LIN {X 0,Y 412.536,Z 861.906,A -85,B 0,C 180,E1 10223.476,E2 10223.476} C_VEL
LIN {X 0,Y 403.903,Z 849.532,A -85,B 0,C 180,E1 10225.593,E2 10225.593} C_VEL
LIN {X 0,Y 401.209,Z 844.898,A -85,B 0,C 180,E1 10226.312,E2 10226.312} C_VEL
LIN {X 0,Y 401.09,Z 843.44,A -85,B 0,C 180,E1 10226.508,E2 10226.508} C_VEL
LIN {X 0,Y 401.209,Z 843.44,A -85,B 0,C 180,E1 10233.172,E2 10233.172} C_VEL
LIN {X 0,Y 401.536,Z 843.44,A -85,B 0,C 180,E1 10240.232,E2 10240.232} C_VEL
LIN {X 0,Y 401.88,Z 843.44,A -85,B 0,C 180,E1 10246.981,E2 10246.981} C_VEL
LIN {X 0,Y 402.092,Z 843.44,A -85,B 0,C 180,E1 10253.536,E2 10253.536} C_VEL
LIN {X 0,Y 402.38,Z 843.44,A -85,B 0,C 180,E1 10260,E2 10260} C_VEL
LIN {X 0,Y 402.145,Z 843.44,A -85,B 0,C 180,E1 10266.464,E2 10266.464} C_VEL
LIN {X 0,Y 401.805,Z 843.44,A -85,B 0,C 180,E1 10273.022,E2 10273.022} C_VEL
LIN {X 0,Y 401.458,Z 843.44,A -85,B 0,C 180,E1 10279.998,E2 10279.998} C_VEL
LIN {X 0,Y 401.24,Z 843.44,A -85,B 0,C 180,E1 10286.827,E2 10286.827} C_VEL
LIN {X 0,Y 401.092,Z 844.186,A -85,B 0,C 180,E1 10293.067,E2 10293.067} C_VEL
LIN {X 0,Y 403.743,Z 849.357,A -85,B 0,C 180,E1 10293.796,E2 10293.796} C_VEL
LIN {X 0,Y 414.864,Z 865.253,A -85,B 0,C 180,E1 10296.457,E2 10296.457} C_VEL
LIN {X 0,Y 433.595,Z 895.537,A -85,B 0,C 180,E1 10300.541,E2 10300.541} C_VEL
LIN {X 0,Y 446.77,Z 923.801,A -85,B 0,C 180,E1 10303.625,E2 10303.625} C_VEL
LIN {X 0,Y 441.038,Z 966.249,A -85,B 0,C 180,E1 10305.53,E2 10305.53} C_VEL
LIN {X 0,Y 433.9,Z 1006.868,A -85,B 0,C 180,E1 10308.269,E2 10308.269} C_VEL
LIN {X 0,Y 425.996,Z 1044.808,A -85,B 0,C 180,E1 10311.841,E2 10311.841} C_VEL
LIN {X 0,Y 418.385,Z 1078.926,A -85,B 0,C 180,E1 10316.189,E2 10316.189} C_VEL
LIN {X 0,Y 411.832,Z 1108.737,A -85,B 0,C 180,E1 10321.255,E2 10321.255} C_VEL
LIN {X 0,Y 406.944,Z 1134.205,A -85,B 0,C 180,E1 10327.086,E2 10327.086} C_VEL
LIN {X 0,Y 404.04,Z 1153.414,A -85,B 0,C 180,E1 10333.175,E2 10333.175} C_VEL
LIN {X 0,Y 403.787,Z 1155.866,A -85,B 0,C 180,E1 10334.164,E2 10334.164} C_VEL
LIN {X 0,Y 400.89,Z 1159.99,A -85,B 0,C 180,E1 10335.894,E2 10335.894} C_VEL
LIN {X 0,Y 395.067,Z 1165.147,A -85,B 0,C 180,E1 10338.532,E2 10338.532} C_VEL
LIN {X 0,Y 394.935,Z 1165.692,A -85,B 0,C 180,E1 10338.841,E2 10338.841} C_VEL
LIN {X 0,Y 394.47,Z 1172.146,A -85,B 0,C 180,E1 10344.029,E2 10344.029} C_VEL
LIN {X 0,Y 394.523,Z 1174.816,A -85,B 0,C 180,E1 10350,E2 10350} C_VEL
LIN {X 0,Y 394.535,Z 1173.409,A -85,B 0,C 180,E1 10354.387,E2 10354.387} C_VEL
LIN {X 0,Y 394.794,Z 1167.57,A -85,B 0,C 180,E1 10359.905,E2 10359.905} C_VEL
LIN {X 0,Y 395.707,Z 1157.209,A -85,B 0,C 180,E1 10365.483,E2 10365.483} C_VEL
LIN {X 0,Y 398.3,Z 1139.989,A -85,B 0,C 180,E1 10371.636,E2 10371.636} C_VEL
LIN {X 0,Y 402.939,Z 1115.912,A -85,B 0,C 180,E1 10377.744,E2 10377.744} C_VEL
LIN {X 0,Y 409.269,Z 1088.112,A -85,B 0,C 180,E1 10382.969,E2 10382.969} C_VEL
LIN {X 0,Y 417.087,Z 1054.957,A -85,B 0,C 180,E1 10387.641,E2 10387.641} C_VEL
LIN {X 0,Y 425.41,Z 1017.824,A -85,B 0,C 180,E1 10391.513,E2 10391.513} C_VEL
LIN {X 0,Y 433.374,Z 977.18,A -85,B 0,C 180,E1 10394.553,E2 10394.553} C_VEL
LIN {X 0,Y 439.964,Z 934.17,A -85,B 0,C 180,E1 10396.732,E2 10396.732} C_VEL
LIN {X 0,Y 440.381,Z 925.23,A -85,B 0,C 180,E1 10397.161,E2 10397.161} C_VEL
LIN {X 0,Y 425.642,Z 894.694,A -85,B 0,C 180,E1 10400.751,E2 10400.751} C_VEL
LIN {X 0,Y 409.009,Z 867.964,A -85,B 0,C 180,E1 10404.593,E2 10404.593} C_VEL
LIN {X 0,Y 396.315,Z 849.753,A -85,B 0,C 180,E1 10407.836,E2 10407.836} C_VEL
LIN {X 0,Y 393.263,Z 844.634,A -85,B 0,C 180,E1 10408.718,E2 10408.718} C_VEL
LIN {X 0,Y 393.154,Z 843.44,A -85,B 0,C 180,E1 10408.818,E2 10408.818} C_VEL
LIN {X 0,Y 393.359,Z 843.44,A -85,B 0,C 180,E1 10415.041,E2 10415.041} C_VEL
LIN {X 0,Y 393.632,Z 843.44,A -85,B 0,C 180,E1 10422.141,E2 10422.141} C_VEL
LIN {X 0,Y 393.836,Z 843.44,A -85,B 0,C 180,E1 10428.955,E2 10428.955} C_VEL
LIN {X 0,Y 394.243,Z 843.44,A -85,B 0,C 180,E1 10435.61,E2 10435.61} C_VEL
LIN {X 0,Y 394.337,Z 843.44,A -85,B 0,C 180,E1 10442.193,E2 10442.193} C_VEL
LIN {X 0,Y 394.018,Z 843.44,A -85,B 0,C 180,E1 10448.811,E2 10448.811} C_VEL
LIN {X 0,Y 393.774,Z 843.44,A -85,B 0,C 180,E1 10455.559,E2 10455.559} C_VEL
LIN {X 0,Y 393.41,Z 843.44,A -85,B 0,C 180,E1 10462.989,E2 10462.989} C_VEL
LIN {X 0,Y 393.294,Z 843.44,A -85,B 0,C 180,E1 10469.919,E2 10469.919} C_VEL
LIN {X 0,Y 393.33,Z 843.44,A -85,B 0,C 180,E1 10471.727,E2 10471.727} C_VEL
LIN {X 0,Y 395.292,Z 848.705,A -85,B 0,C 180,E1 10472.377,E2 10472.377} C_VEL
LIN {X 0,Y 398.335,Z 852.335,A -85,B 0,C 180,E1 10473.186,E2 10473.186} C_VEL
LIN {X 0,Y 414.19,Z 876.466,A -85,B 0,C 180,E1 10477.277,E2 10477.277} C_VEL
LIN {X 0,Y 429.429,Z 905.007,A -85,B 0,C 180,E1 10481.288,E2 10481.288} C_VEL
LIN {X 0,Y 438.439,Z 927.966,A -85,B 0,C 180,E1 10484.052,E2 10484.052} C_VEL
LIN {X 0,Y 431.611,Z 968.432,A -85,B 0,C 180,E1 10486.494,E2 10486.494} C_VEL
LIN {X 0,Y 423.482,Z 1006.655,A -85,B 0,C 180,E1 10489.77,E2 10489.77} C_VEL
LIN {X 0,Y 415.09,Z 1041.89,A -85,B 0,C 180,E1 10493.94,E2 10493.94} C_VEL
LIN {X 0,Y 407.221,Z 1073.607,A -85,B 0,C 180,E1 10499.059,E2 10499.059} C_VEL
LIN {X 0,Y 401.372,Z 1098.435,A -85,B 0,C 180,E1 10504.459,E2 10504.459} C_VEL
LIN {X 0,Y 397.287,Z 1119.022,A -85,B 0,C 180,E1 10510.615,E2 10510.615} C_VEL
LIN {X 0,Y 395.387,Z 1133.199,A -85,B 0,C 180,E1 10516.762,E2 10516.762} C_VEL
LIN {X 0,Y 394.56,Z 1141.136,A -85,B 0,C 180,E1 10522.307,E2 10522.307} C_VEL
LIN {X 0,Y 394.48,Z 1144.909,A -85,B 0,C 180,E1 10527.807,E2 10527.807} C_VEL
LIN {X 0,Y 394.579,Z 1144.88,A -85,B 0,C 180,E1 10532.192,E2 10532.192} C_VEL
LIN {X 0,Y 394.625,Z 1141.038,A -85,B 0,C 180,E1 10537.691,E2 10537.691} C_VEL
LIN {X 0,Y 395.504,Z 1132.152,A -85,B 0,C 180,E1 10543.672,E2 10543.672} C_VEL
LIN {X 0,Y 397.375,Z 1118.609,A -85,B 0,C 180,E1 10549.449,E2 10549.449} C_VEL
LIN {X 0,Y 401.431,Z 1098.022,A -85,B 0,C 180,E1 10555.559,E2 10555.559} C_VEL
LIN {X 0,Y 407.649,Z 1071.682,A -85,B 0,C 180,E1 10561.214,E2 10561.214} C_VEL
LIN {X 0,Y 415.306,Z 1041.141,A -85,B 0,C 180,E1 10566.063,E2 10566.063} C_VEL
LIN {X 0,Y 423.441,Z 1006.999,A -85,B 0,C 180,E1 10570.1,E2 10570.1} C_VEL
LIN {X 0,Y 431.425,Z 969.351,A -85,B 0,C 180,E1 10573.35,E2 10573.35} C_VEL
LIN {X 0,Y 438.451,Z 927.099,A -85,B 0,C 180,E1 10575.909,E2 10575.909} C_VEL
LIN {X 0,Y 424.695,Z 895.119,A -85,B 0,C 180,E1 10579.911,E2 10579.911} C_VEL
LIN {X 0,Y 408.354,Z 867.268,A -85,B 0,C 180,E1 10584.097,E2 10584.097} C_VEL
LIN {X 0,Y 396.169,Z 849.642,A -85,B 0,C 180,E1 10587.277,E2 10587.277} C_VEL
LIN {X 0,Y 393.281,Z 844.581,A -85,B 0,C 180,E1 10588.118,E2 10588.118} C_VEL
LIN {X 0,Y 393.187,Z 843.44,A -85,B 0,C 180,E1 10588.384,E2 10588.384} C_VEL
LIN {X 0,Y 393.352,Z 843.44,A -85,B 0,C 180,E1 10595.041,E2 10595.041} C_VEL
LIN {X 0,Y 393.712,Z 843.44,A -85,B 0,C 180,E1 10602.145,E2 10602.145} C_VEL
LIN {X 0,Y 393.997,Z 843.44,A -85,B 0,C 180,E1 10608.96,E2 10608.96} C_VEL
LIN {X 0,Y 394.278,Z 843.44,A -85,B 0,C 180,E1 10615.61,E2 10615.61} C_VEL
LIN {X 0,Y 394.482,Z 843.44,A -85,B 0,C 180,E1 10622.192,E2 10622.192} C_VEL
LIN {X 0,Y 394.04,Z 843.44,A -85,B 0,C 180,E1 10628.811,E2 10628.811} C_VEL
LIN {X 0,Y 393.727,Z 843.44,A -85,B 0,C 180,E1 10635.562,E2 10635.562} C_VEL
LIN {X 0,Y 393.413,Z 843.44,A -85,B 0,C 180,E1 10642.991,E2 10642.991} C_VEL
LIN {X 0,Y 393.194,Z 843.44,A -85,B 0,C 180,E1 10649.927,E2 10649.927} C_VEL
LIN {X 0,Y 393.158,Z 843.44,A -85,B 0,C 180,E1 10651.238,E2 10651.238} C_VEL
LIN {X 0,Y 395.313,Z 848.816,A -85,B 0,C 180,E1 10651.927,E2 10651.927} C_VEL
LIN {X 0,Y 398.159,Z 852.24,A -85,B 0,C 180,E1 10652.683,E2 10652.683} C_VEL
LIN {X 0,Y 417.725,Z 881.071,A -85,B 0,C 180,E1 10657.445,E2 10657.445} C_VEL
LIN {X 0,Y 434.757,Z 912.535,A -85,B 0,C 180,E1 10661.424,E2 10661.424} C_VEL
LIN {X 0,Y 440.859,Z 927.31,A -85,B 0,C 180,E1 10663.022,E2 10663.022} C_VEL
LIN {X 0,Y 435.214,Z 966.606,A -85,B 0,C 180,E1 10664.827,E2 10664.827} C_VEL
LIN {X 0,Y 427.789,Z 1006.919,A -85,B 0,C 180,E1 10667.575,E2 10667.575} C_VEL
LIN {X 0,Y 419.756,Z 1043.593,A -85,B 0,C 180,E1 10671.047,E2 10671.047} C_VEL
LIN {X 0,Y 411.516,Z 1078.613,A -85,B 0,C 180,E1 10675.546,E2 10675.546} C_VEL
LIN {X 0,Y 404.609,Z 1108.428,A -85,B 0,C 180,E1 10680.692,E2 10680.692} C_VEL
LIN {X 0,Y 399.343,Z 1133.895,A -85,B 0,C 180,E1 10686.624,E2 10686.624} C_VEL
LIN {X 0,Y 396.253,Z 1153.109,A -85,B 0,C 180,E1 10692.835,E2 10692.835} C_VEL
LIN {X 0,Y 394.935,Z 1165.692,A -85,B 0,C 180,E1 10698.841,E2 10698.841} C_VEL
LIN {X 0,Y 392.233,Z 1168.533,A -85,B 0,C 180,E1 10700.665,E2 10700.665} C_VEL
LIN {X 0,Y 386.689,Z 1171.487,A -85,B 0,C 180,E1 10703.446,E2 10703.446} C_VEL
LIN {X 0,Y 386.568,Z 1171.734,A -85,B 0,C 180,E1 10703.771,E2 10703.771} C_VEL
LIN {X 0,Y 386.572,Z 1174.166,A -85,B 0,C 180,E1 10707.763,E2 10707.763} C_VEL
LIN {X 0,Y 386.751,Z 1174.172,A -85,B 0,C 180,E1 10712.236,E2 10712.236} C_VEL
LIN {X 0,Y 386.706,Z 1170.117,A -85,B 0,C 180,E1 10717.85,E2 10717.85} C_VEL
LIN {X 0,Y 387.441,Z 1161.671,A -85,B 0,C 180,E1 10723.515,E2 10723.515} C_VEL
LIN {X 0,Y 389.437,Z 1146.627,A -85,B 0,C 180,E1 10729.819,E2 10729.819} C_VEL
LIN {X 0,Y 393.295,Z 1126.005,A -85,B 0,C 180,E1 10735.858,E2 10735.858} C_VEL
LIN {X 0,Y 399.461,Z 1099.256,A -85,B 0,C 180,E1 10741.611,E2 10741.611} C_VEL
LIN {X 0,Y 407.687,Z 1066.369,A -85,B 0,C 180,E1 10746.83,E2 10746.83} C_VEL
LIN {X 0,Y 416.394,Z 1030.711,A -85,B 0,C 180,E1 10750.997,E2 10750.997} C_VEL
LIN {X 0,Y 424.702,Z 992.738,A -85,B 0,C 180,E1 10754.24,E2 10754.24} C_VEL
LIN {X 0,Y 431.692,Z 953.938,A -85,B 0,C 180,E1 10756.581,E2 10756.581} C_VEL
LIN {X 0,Y 434.563,Z 928.474,A -85,B 0,C 180,E1 10757.795,E2 10757.795} C_VEL
LIN {X 0,Y 420.517,Z 898.817,A -85,B 0,C 180,E1 10761.43,E2 10761.43} C_VEL
LIN {X 0,Y 404.771,Z 873.027,A -85,B 0,C 180,E1 10765.284,E2 10765.284} C_VEL
LIN {X 0,Y 392.687,Z 855.818,A -85,B 0,C 180,E1 10768.473,E2 10768.473} C_VEL
LIN {X 0,Y 388.57,Z 849.833,A -85,B 0,C 180,E1 10769.679,E2 10769.679} C_VEL
LIN {X 0,Y 385.501,Z 845.356,A -85,B 0,C 180,E1 10770.626,E2 10770.626} C_VEL
LIN {X 0,Y 385.254,Z 843.44,A -85,B 0,C 180,E1 10770.85,E2 10770.85} C_VEL
LIN {X 0,Y 385.514,Z 843.44,A -85,B 0,C 180,E1 10776.957,E2 10776.957} C_VEL
LIN {X 0,Y 385.745,Z 843.44,A -85,B 0,C 180,E1 10784.108,E2 10784.108} C_VEL
LIN {X 0,Y 386.034,Z 843.44,A -85,B 0,C 180,E1 10791.004,E2 10791.004} C_VEL
LIN {X 0,Y 386.575,Z 843.44,A -85,B 0,C 180,E1 10797.763,E2 10797.763} C_VEL
LIN {X 0,Y 386.362,Z 843.44,A -85,B 0,C 180,E1 10804.48,E2 10804.48} C_VEL
LIN {X 0,Y 386.024,Z 843.44,A -85,B 0,C 180,E1 10811.271,E2 10811.271} C_VEL
LIN {X 0,Y 385.695,Z 843.44,A -85,B 0,C 180,E1 10818.239,E2 10818.239} C_VEL
LIN {X 0,Y 385.366,Z 843.44,A -85,B 0,C 180,E1 10825.758,E2 10825.758} C_VEL
LIN {X 0,Y 385.373,Z 843.44,A -85,B 0,C 180,E1 10829.752,E2 10829.752} C_VEL
LIN {X 0,Y 387.473,Z 848.827,A -85,B 0,C 180,E1 10830.491,E2 10830.491} C_VEL
LIN {X 0,Y 390.513,Z 852.225,A -85,B 0,C 180,E1 10831.366,E2 10831.366} C_VEL
LIN {X 0,Y 406.881,Z 876.641,A -85,B 0,C 180,E1 10835.891,E2 10835.891} C_VEL
LIN {X 0,Y 422.767,Z 906.139,A -85,B 0,C 180,E1 10840.296,E2 10840.296} C_VEL
LIN {X 0,Y 432.571,Z 930.558,A -85,B 0,C 180,E1 10843.415,E2 10843.415} C_VEL
LIN {X 0,Y 425.827,Z 968.818,A -85,B 0,C 180,E1 10845.759,E2 10845.759} C_VEL
LIN {X 0,Y 417.032,Z 1008.301,A -85,B 0,C 180,E1 10849.19,E2 10849.19} C_VEL
LIN {X 0,Y 408.103,Z 1043.878,A -85,B 0,C 180,E1 10853.513,E2 10853.513} C_VEL
LIN {X 0,Y 400.196,Z 1073.911,A -85,B 0,C 180,E1 10858.454,E2 10858.454} C_VEL
LIN {X 0,Y 394.079,Z 1098.735,A -85,B 0,C 180,E1 10863.951,E2 10863.951} C_VEL
LIN {X 0,Y 389.646,Z 1119.254,A -85,B 0,C 180,E1 10870.192,E2 10870.192} C_VEL
LIN {X 0,Y 387.567,Z 1133.498,A -85,B 0,C 180,E1 10876.49,E2 10876.49} C_VEL
LIN {X 0,Y 386.683,Z 1141.433,A -85,B 0,C 180,E1 10882.149,E2 10882.149} C_VEL
LIN {X 0,Y 386.581,Z 1145.206,A -85,B 0,C 180,E1 10887.763,E2 10887.763} C_VEL
LIN {X 0,Y 386.678,Z 1145.177,A -85,B 0,C 180,E1 10892.236,E2 10892.236} C_VEL
LIN {X 0,Y 386.745,Z 1141.337,A -85,B 0,C 180,E1 10897.849,E2 10897.849} C_VEL
LIN {X 0,Y 387.634,Z 1133.323,A -85,B 0,C 180,E1 10903.507,E2 10903.507} C_VEL
LIN {X 0,Y 389.689,Z 1119.028,A -85,B 0,C 180,E1 10909.805,E2 10909.805} C_VEL
LIN {X 0,Y 394.081,Z 1098.332,A -85,B 0,C 180,E1 10916.071,E2 10916.071} C_VEL
LIN {X 0,Y 400.688,Z 1071.993,A -85,B 0,C 180,E1 10921.819,E2 10921.819} C_VEL
LIN {X 0,Y 408.657,Z 1041.936,A -85,B 0,C 180,E1 10926.668,E2 10926.668} C_VEL
LIN {X 0,Y 417.257,Z 1007.566,A -85,B 0,C 180,E1 10930.786,E2 10930.786} C_VEL
LIN {X 0,Y 425.671,Z 969.676,A -85,B 0,C 180,E1 10934.084,E2 10934.084} C_VEL
LIN {X 0,Y 432.479,Z 930.241,A -85,B 0,C 180,E1 10936.527,E2 10936.527} C_VEL
LIN {X 0,Y 419.451,Z 899.303,A -85,B 0,C 180,E1 10940.567,E2 10940.567} C_VEL
LIN {X 0,Y 402.739,Z 869.859,A -85,B 0,C 180,E1 10945.135,E2 10945.135} C_VEL
LIN {X 0,Y 388.559,Z 849.846,A -85,B 0,C 180,E1 10949.081,E2 10949.081} C_VEL
LIN {X 0,Y 385.437,Z 844.892,A -85,B 0,C 180,E1 10950.056,E2 10950.056} C_VEL
LIN {X 0,Y 385.275,Z 843.44,A -85,B 0,C 180,E1 10950.366,E2 10950.366} C_VEL
LIN {X 0,Y 385.51,Z 843.44,A -85,B 0,C 180,E1 10956.958,E2 10956.958} C_VEL
LIN {X 0,Y 385.91,Z 843.44,A -85,B 0,C 180,E1 10964.115,E2 10964.115} C_VEL
LIN {X 0,Y 386.126,Z 843.44,A -85,B 0,C 180,E1 10971.007,E2 10971.007} C_VEL
LIN {X 0,Y 386.439,Z 843.44,A -85,B 0,C 180,E1 10977.762,E2 10977.762} C_VEL
LIN {X 0,Y 386.335,Z 843.44,A -85,B 0,C 180,E1 10984.481,E2 10984.481} C_VEL
LIN {X 0,Y 385.981,Z 843.44,A -85,B 0,C 180,E1 10991.272,E2 10991.272} C_VEL
LIN {X 0,Y 385.668,Z 843.44,A -85,B 0,C 180,E1 10998.241,E2 10998.241} C_VEL
LIN {X 0,Y 385.383,Z 843.44,A -85,B 0,C 180,E1 11005.512,E2 11005.512} C_VEL
LIN {X 0,Y 385.302,Z 844.197,A -85,B 0,C 180,E1 11009.31,E2 11009.31} C_VEL
LIN {X 0,Y 388.071,Z 849.476,A -85,B 0,C 180,E1 11010.212,E2 11010.212} C_VEL
LIN {X 0,Y 390.458,Z 852.409,A -85,B 0,C 180,E1 11010.903,E2 11010.903} C_VEL
LIN {X 0,Y 407.64,Z 877.287,A -85,B 0,C 180,E1 11015.444,E2 11015.444} C_VEL
LIN {X 0,Y 424.478,Z 906.09,A -85,B 0,C 180,E1 11019.534,E2 11019.534} C_VEL
LIN {X 0,Y 434.994,Z 930.293,A -85,B 0,C 180,E1 11022.373,E2 11022.373} C_VEL
LIN {X 0,Y 428.859,Z 970.174,A -85,B 0,C 180,E1 11024.293,E2 11024.293} C_VEL
LIN {X 0,Y 421.471,Z 1008.185,A -85,B 0,C 180,E1 11026.964,E2 11026.964} C_VEL
LIN {X 0,Y 412.982,Z 1044.955,A -85,B 0,C 180,E1 11030.521,E2 11030.521} C_VEL
LIN {X 0,Y 404.635,Z 1078.785,A -85,B 0,C 180,E1 11034.963,E2 11034.963} C_VEL
LIN {X 0,Y 397.422,Z 1108.117,A -85,B 0,C 180,E1 11040.109,E2 11040.109} C_VEL
LIN {X 0,Y 391.775,Z 1133.585,A -85,B 0,C 180,E1 11046.145,E2 11046.145} C_VEL
LIN {X 0,Y 388.705,Z 1151.329,A -85,B 0,C 180,E1 11051.906,E2 11051.906} C_VEL
LIN {X 0,Y 387.252,Z 1163.986,A -85,B 0,C 180,E1 11057.801,E2 11057.801} C_VEL
LIN {X 0,Y 386.629,Z 1171.345,A -85,B 0,C 180,E1 11063.276,E2 11063.276} C_VEL
LIN {X 0,Y 386.568,Z 1171.734,A -85,B 0,C 180,E1 11063.771,E2 11063.771} C_VEL
LIN {X 0,Y 383.964,Z 1173.1,A -85,B 0,C 180,E1 11065.669,E2 11065.669} C_VEL
LIN {X 0,Y 378.708,Z 1174.007,A -85,B 0,C 180,E1 11068.538,E2 11068.538} C_VEL
LIN {X 0,Y 378.626,Z 1174.048,A -85,B 0,C 180,E1 11068.871,E2 11068.871} C_VEL
LIN {X 0,Y 378.845,Z 1173.876,A -85,B 0,C 180,E1 11072.283,E2 11072.283} C_VEL
LIN {X 0,Y 378.821,Z 1169.818,A -85,B 0,C 180,E1 11078.015,E2 11078.015} C_VEL
LIN {X 0,Y 379.571,Z 1161.367,A -85,B 0,C 180,E1 11083.8,E2 11083.8} C_VEL
LIN {X 0,Y 381.744,Z 1146.32,A -85,B 0,C 180,E1 11090.236,E2 11090.236} C_VEL
LIN {X 0,Y 386.289,Z 1124.406,A -85,B 0,C 180,E1 11096.719,E2 11096.719} C_VEL
LIN {X 0,Y 392.864,Z 1097.403,A -85,B 0,C 180,E1 11102.531,E2 11102.531} C_VEL
LIN {X 0,Y 401.145,Z 1066.056,A -85,B 0,C 180,E1 11107.534,E2 11107.534} C_VEL
LIN {X 0,Y 410.439,Z 1029.58,A -85,B 0,C 180,E1 11111.828,E2 11111.828} C_VEL
LIN {X 0,Y 419.296,Z 990.383,A -85,B 0,C 180,E1 11115.164,E2 11115.164} C_VEL
LIN {X 0,Y 426.852,Z 949.888,A -85,B 0,C 180,E1 11117.556,E2 11117.556} C_VEL
LIN {X 0,Y 428.835,Z 931.703,A -85,B 0,C 180,E1 11118.443,E2 11118.443} C_VEL
LIN {X 0,Y 414.799,Z 901.66,A -85,B 0,C 180,E1 11122.294,E2 11122.294} C_VEL
LIN {X 0,Y 398.816,Z 875.264,A -85,B 0,C 180,E1 11126.451,E2 11126.451} C_VEL
LIN {X 0,Y 385.116,Z 856.082,A -85,B 0,C 180,E1 11130.331,E2 11130.331} C_VEL
LIN {X 0,Y 381.085,Z 850.146,A -85,B 0,C 180,E1 11131.63,E2 11131.63} C_VEL
LIN {X 0,Y 377.608,Z 845.437,A -85,B 0,C 180,E1 11132.803,E2 11132.803} C_VEL
LIN {X 0,Y 377.364,Z 843.44,A -85,B 0,C 180,E1 11133.105,E2 11133.105} C_VEL
LIN {X 0,Y 377.637,Z 843.44,A -85,B 0,C 180,E1 11138.923,E2 11138.923} C_VEL
LIN {X 0,Y 377.882,Z 843.44,A -85,B 0,C 180,E1 11146.137,E2 11146.137} C_VEL
LIN {X 0,Y 378.33,Z 843.44,A -85,B 0,C 180,E1 11153.128,E2 11153.128} C_VEL
LIN {X 0,Y 378.628,Z 843.44,A -85,B 0,C 180,E1 11160,E2 11160} C_VEL
LIN {X 0,Y 378.323,Z 843.44,A -85,B 0,C 180,E1 11166.872,E2 11166.872} C_VEL
LIN {X 0,Y 378.021,Z 843.44,A -85,B 0,C 180,E1 11173.857,E2 11173.857} C_VEL
LIN {X 0,Y 377.633,Z 843.44,A -85,B 0,C 180,E1 11181.077,E2 11181.077} C_VEL
LIN {X 0,Y 377.427,Z 843.515,A -85,B 0,C 180,E1 11187.549,E2 11187.549} C_VEL
LIN {X 0,Y 379.422,Z 848.673,A -85,B 0,C 180,E1 11188.331,E2 11188.331} C_VEL
LIN {X 0,Y 382.7,Z 852.12,A -85,B 0,C 180,E1 11189.367,E2 11189.367} C_VEL
LIN {X 0,Y 397.567,Z 873.908,A -85,B 0,C 180,E1 11193.826,E2 11193.826} C_VEL
LIN {X 0,Y 412.618,Z 900.242,A -85,B 0,C 180,E1 11198.189,E2 11198.189} C_VEL
LIN {X 0,Y 424.836,Z 928.377,A -85,B 0,C 180,E1 11202.099,E2 11202.099} C_VEL
LIN {X 0,Y 426.507,Z 934.531,A -85,B 0,C 180,E1 11202.833,E2 11202.833} C_VEL
LIN {X 0,Y 419.384,Z 972.555,A -85,B 0,C 180,E1 11205.26,E2 11205.26} C_VEL
LIN {X 0,Y 410.623,Z 1009.825,A -85,B 0,C 180,E1 11208.586,E2 11208.586} C_VEL
LIN {X 0,Y 401.559,Z 1044.313,A -85,B 0,C 180,E1 11212.843,E2 11212.843} C_VEL
LIN {X 0,Y 393.263,Z 1074.214,A -85,B 0,C 180,E1 11217.831,E2 11217.831} C_VEL
LIN {X 0,Y 386.735,Z 1099.222,A -85,B 0,C 180,E1 11223.472,E2 11223.472} C_VEL
LIN {X 0,Y 382.038,Z 1119.556,A -85,B 0,C 180,E1 11229.78,E2 11229.78} C_VEL
LIN {X 0,Y 379.777,Z 1133.797,A -85,B 0,C 180,E1 11236.207,E2 11236.207} C_VEL
LIN {X 0,Y 378.804,Z 1141.731,A -85,B 0,C 180,E1 11241.985,E2 11241.985} C_VEL
LIN {X 0,Y 378.682,Z 1145.502,A -85,B 0,C 180,E1 11247.716,E2 11247.716} C_VEL
LIN {X 0,Y 378.777,Z 1145.474,A -85,B 0,C 180,E1 11252.283,E2 11252.283} C_VEL
LIN {X 0,Y 378.889,Z 1141.636,A -85,B 0,C 180,E1 11258.013,E2 11258.013} C_VEL
LIN {X 0,Y 379.827,Z 1133.626,A -85,B 0,C 180,E1 11263.79,E2 11263.79} C_VEL
LIN {X 0,Y 382.049,Z 1119.335,A -85,B 0,C 180,E1 11270.219,E2 11270.219} C_VEL
LIN {X 0,Y 386.505,Z 1099.673,A -85,B 0,C 180,E1 11276.324,E2 11276.324} C_VEL
LIN {X 0,Y 393.373,Z 1073.813,A -85,B 0,C 180,E1 11282.158,E2 11282.158} C_VEL
LIN {X 0,Y 402.097,Z 1042.502,A -85,B 0,C 180,E1 11287.324,E2 11287.324} C_VEL
LIN {X 0,Y 411.179,Z 1007.885,A -85,B 0,C 180,E1 11291.519,E2 11291.519} C_VEL
LIN {X 0,Y 419.968,Z 969.983,A -85,B 0,C 180,E1 11294.842,E2 11294.842} C_VEL
LIN {X 0,Y 426.377,Z 933.046,A -85,B 0,C 180,E1 11297.206,E2 11297.206} C_VEL
LIN {X 0,Y 413.914,Z 902.607,A -85,B 0,C 180,E1 11301.33,E2 11301.33} C_VEL
LIN {X 0,Y 398.105,Z 874.851,A -85,B 0,C 180,E1 11305.899,E2 11305.899} C_VEL
LIN {X 0,Y 385.288,Z 856.281,A -85,B 0,C 180,E1 11309.677,E2 11309.677} C_VEL
LIN {X 0,Y 380.858,Z 850.005,A -85,B 0,C 180,E1 11311.092,E2 11311.092} C_VEL
LIN {X 0,Y 377.529,Z 844.979,A -85,B 0,C 180,E1 11312.234,E2 11312.234} C_VEL
LIN {X 0,Y 377.349,Z 843.44,A -85,B 0,C 180,E1 11312.392,E2 11312.392} C_VEL
LIN {X 0,Y 377.644,Z 843.44,A -85,B 0,C 180,E1 11318.924,E2 11318.924} C_VEL
LIN {X 0,Y 378.07,Z 843.44,A -85,B 0,C 180,E1 11326.145,E2 11326.145} C_VEL
LIN {X 0,Y 378.328,Z 843.44,A -85,B 0,C 180,E1 11333.128,E2 11333.128} C_VEL
LIN {X 0,Y 378.673,Z 843.44,A -85,B 0,C 180,E1 11340,E2 11340} C_VEL
LIN {X 0,Y 378.402,Z 843.44,A -85,B 0,C 180,E1 11346.871,E2 11346.871} C_VEL
LIN {X 0,Y 377.956,Z 843.44,A -85,B 0,C 180,E1 11353.86,E2 11353.86} C_VEL
LIN {X 0,Y 377.622,Z 843.44,A -85,B 0,C 180,E1 11361.078,E2 11361.078} C_VEL
LIN {X 0,Y 377.42,Z 844.229,A -85,B 0,C 180,E1 11367.131,E2 11367.131} C_VEL
LIN {X 0,Y 380.045,Z 849.339,A -85,B 0,C 180,E1 11368.084,E2 11368.084} C_VEL
LIN {X 0,Y 382.648,Z 852.309,A -85,B 0,C 180,E1 11368.91,E2 11368.91} C_VEL
LIN {X 0,Y 397.159,Z 872.998,A -85,B 0,C 180,E1 11373.133,E2 11373.133} C_VEL
LIN {X 0,Y 413.401,Z 899.125,A -85,B 0,C 180,E1 11377.361,E2 11377.361} C_VEL
LIN {X 0,Y 427.986,Z 929.72,A -85,B 0,C 180,E1 11381.324,E2 11381.324} C_VEL
LIN {X 0,Y 429.039,Z 934.674,A -85,B 0,C 180,E1 11381.764,E2 11381.764} C_VEL
LIN {X 0,Y 421.653,Z 978.391,A -85,B 0,C 180,E1 11384.019,E2 11384.019} C_VEL
LIN {X 0,Y 412.864,Z 1019.432,A -85,B 0,C 180,E1 11387.198,E2 11387.198} C_VEL
LIN {X 0,Y 403.964,Z 1055.351,A -85,B 0,C 180,E1 11391.063,E2 11391.063} C_VEL
LIN {X 0,Y 395.033,Z 1089.295,A -85,B 0,C 180,E1 11396.036,E2 11396.036} C_VEL
LIN {X 0,Y 388.028,Z 1116.746,A -85,B 0,C 180,E1 11401.441,E2 11401.441} C_VEL
LIN {X 0,Y 382.955,Z 1140.091,A -85,B 0,C 180,E1 11407.688,E2 11407.688} C_VEL
LIN {X 0,Y 380.182,Z 1156.604,A -85,B 0,C 180,E1 11413.869,E2 11413.869} C_VEL
LIN {X 0,Y 379.018,Z 1166.97,A -85,B 0,C 180,E1 11419.679,E2 11419.679} C_VEL
LIN {X 0,Y 378.696,Z 1172.813,A -85,B 0,C 180,E1 11425.429,E2 11425.429} C_VEL
LIN {X 0,Y 378.626,Z 1174.048,A -85,B 0,C 180,E1 11428.871,E2 11428.871} C_VEL
LIN {X 0,Y 376.16,Z 1174.04,A -85,B 0,C 180,E1 11430.831,E2 11430.831} C_VEL
LIN {X 0,Y 370.82,Z 1172.766,A -85,B 0,C 180,E1 11434.122,E2 11434.122} C_VEL
LIN {X 0,Y 371.036,Z 1168.266,A -85,B 0,C 180,E1 11439.363,E2 11439.363} C_VEL
LIN {X 0,Y 372.167,Z 1157.538,A -85,B 0,C 180,E1 11445.884,E2 11445.884} C_VEL
LIN {X 0,Y 375.062,Z 1141.279,A -85,B 0,C 180,E1 11452.28,E2 11452.28} C_VEL
LIN {X 0,Y 380.011,Z 1119.297,A -85,B 0,C 180,E1 11458.458,E2 11458.458} C_VEL
LIN {X 0,Y 386.797,Z 1093.853,A -85,B 0,C 180,E1 11463.776,E2 11463.776} C_VEL
LIN {X 0,Y 395.109,Z 1063.973,A -85,B 0,C 180,E1 11468.502,E2 11468.502} C_VEL
LIN {X 0,Y 404.477,Z 1028.861,A -85,B 0,C 180,E1 11472.642,E2 11472.642} C_VEL
LIN {X 0,Y 413.669,Z 989.935,A -85,B 0,C 180,E1 11475.968,E2 11475.968} C_VEL
LIN {X 0,Y 421.657,Z 948.183,A -85,B 0,C 180,E1 11478.431,E2 11478.431} C_VEL
LIN {X 0,Y 423.436,Z 935.798,A -85,B 0,C 180,E1 11479.011,E2 11479.011} C_VEL
LIN {X 0,Y 410,Z 906.276,A -85,B 0,C 180,E1 11482.939,E2 11482.939} C_VEL
LIN {X 0,Y 395.064,Z 881.076,A -85,B 0,C 180,E1 11487.047,E2 11487.047} C_VEL
LIN {X 0,Y 381.653,Z 861.918,A -85,B 0,C 180,E1 11491.027,E2 11491.027} C_VEL
LIN {X 0,Y 377.311,Z 856.085,A -85,B 0,C 180,E1 11492.461,E2 11492.461} C_VEL
LIN {X 0,Y 373.359,Z 850.218,A -85,B 0,C 180,E1 11493.883,E2 11493.883} C_VEL
LIN {X 0,Y 369.785,Z 845.578,A -85,B 0,C 180,E1 11495.231,E2 11495.231} C_VEL
LIN {X 0,Y 369.521,Z 843.44,A -85,B 0,C 180,E1 11495.441,E2 11495.441} C_VEL
LIN {X 0,Y 369.774,Z 843.44,A -85,B 0,C 180,E1 11500.946,E2 11500.946} C_VEL
LIN {X 0,Y 370.042,Z 843.44,A -85,B 0,C 180,E1 11508.235,E2 11508.235} C_VEL
LIN {X 0,Y 370.506,Z 843.44,A -85,B 0,C 180,E1 11515.328,E2 11515.328} C_VEL
LIN {X 0,Y 370.751,Z 843.44,A -85,B 0,C 180,E1 11520,E2 11520} C_VEL
LIN {X 0,Y 370.392,Z 843.44,A -85,B 0,C 180,E1 11527.02,E2 11527.02} C_VEL
LIN {X 0,Y 370.095,Z 843.44,A -85,B 0,C 180,E1 11534.16,E2 11534.16} C_VEL
LIN {X 0,Y 369.693,Z 843.44,A -85,B 0,C 180,E1 11541.552,E2 11541.552} C_VEL
LIN {X 0,Y 369.519,Z 843.756,A -85,B 0,C 180,E1 11545.081,E2 11545.081} C_VEL
LIN {X 0,Y 371.586,Z 848.762,A -85,B 0,C 180,E1 11545.98,E2 11545.98} C_VEL
LIN {X 0,Y 374.98,Z 852.27,A -85,B 0,C 180,E1 11547.181,E2 11547.181} C_VEL
LIN {X 0,Y 389.017,Z 872.069,A -85,B 0,C 180,E1 11551.782,E2 11551.782} C_VEL
LIN {X 0,Y 404.476,Z 898.403,A -85,B 0,C 180,E1 11556.565,E2 11556.565} C_VEL
LIN {X 0,Y 417.261,Z 927.021,A -85,B 0,C 180,E1 11560.807,E2 11560.807} C_VEL
LIN {X 0,Y 420.817,Z 936.747,A -85,B 0,C 180,E1 11562.144,E2 11562.144} C_VEL
LIN {X 0,Y 413.725,Z 972.849,A -85,B 0,C 180,E1 11564.478,E2 11564.478} C_VEL
LIN {X 0,Y 404.63,Z 1010.121,A -85,B 0,C 180,E1 11567.833,E2 11567.833} C_VEL
LIN {X 0,Y 395.354,Z 1043.94,A -85,B 0,C 180,E1 11572.035,E2 11572.035} C_VEL
LIN {X 0,Y 386.278,Z 1074.783,A -85,B 0,C 180,E1 11577.239,E2 11577.239} C_VEL
LIN {X 0,Y 379.234,Z 1100.267,A -85,B 0,C 180,E1 11583.129,E2 11583.129} C_VEL
LIN {X 0,Y 374.426,Z 1119.858,A -85,B 0,C 180,E1 11589.351,E2 11589.351} C_VEL
LIN {X 0,Y 371.973,Z 1134.097,A -85,B 0,C 180,E1 11595.912,E2 11595.912} C_VEL
LIN {X 0,Y 370.952,Z 1142.027,A -85,B 0,C 180,E1 11601.814,E2 11601.814} C_VEL
LIN {X 0,Y 370.811,Z 1145.797,A -85,B 0,C 180,E1 11607.667,E2 11607.667} C_VEL
LIN {X 0,Y 370.9,Z 1145.77,A -85,B 0,C 180,E1 11612.331,E2 11612.331} C_VEL
LIN {X 0,Y 371.028,Z 1141.935,A -85,B 0,C 180,E1 11618.184,E2 11618.184} C_VEL
LIN {X 0,Y 372.005,Z 1133.931,A -85,B 0,C 180,E1 11624.086,E2 11624.086} C_VEL
LIN {X 0,Y 374.438,Z 1119.642,A -85,B 0,C 180,E1 11630.648,E2 11630.648} C_VEL
LIN {X 0,Y 379.622,Z 1098.738,A -85,B 0,C 180,E1 11637.202,E2 11637.202} C_VEL
LIN {X 0,Y 386.958,Z 1072.61,A -85,B 0,C 180,E1 11643.09,E2 11643.09} C_VEL
LIN {X 0,Y 395.837,Z 1042.227,A -85,B 0,C 180,E1 11648.117,E2 11648.117} C_VEL
LIN {X 0,Y 405.423,Z 1007.203,A -85,B 0,C 180,E1 11652.374,E2 11652.374} C_VEL
LIN {X 0,Y 414.343,Z 970.289,A -85,B 0,C 180,E1 11655.621,E2 11655.621} C_VEL
LIN {X 0,Y 420.446,Z 936.088,A -85,B 0,C 180,E1 11657.869,E2 11657.869} C_VEL
LIN {X 0,Y 408.636,Z 906.856,A -85,B 0,C 180,E1 11662.003,E2 11662.003} C_VEL
LIN {X 0,Y 394.232,Z 880.671,A -85,B 0,C 180,E1 11666.454,E2 11666.454} C_VEL
LIN {X 0,Y 382.163,Z 862.709,A -85,B 0,C 180,E1 11670.23,E2 11670.23} C_VEL
LIN {X 0,Y 377.344,Z 856.147,A -85,B 0,C 180,E1 11671.839,E2 11671.839} C_VEL
LIN {X 0,Y 373.38,Z 850.266,A -85,B 0,C 180,E1 11673.26,E2 11673.26} C_VEL
LIN {X 0,Y 369.701,Z 845.297,A -85,B 0,C 180,E1 11674.652,E2 11674.652} C_VEL
LIN {X 0,Y 369.476,Z 843.44,A -85,B 0,C 180,E1 11674.981,E2 11674.981} C_VEL
LIN {X 0,Y 369.824,Z 843.44,A -85,B 0,C 180,E1 11680.949,E2 11680.949} C_VEL
LIN {X 0,Y 370.224,Z 843.44,A -85,B 0,C 180,E1 11688.242,E2 11688.242} C_VEL
LIN {X 0,Y 370.537,Z 843.44,A -85,B 0,C 180,E1 11695.328,E2 11695.328} C_VEL
LIN {X 0,Y 370.755,Z 843.44,A -85,B 0,C 180,E1 11702.333,E2 11702.333} C_VEL
LIN {X 0,Y 370.238,Z 843.44,A -85,B 0,C 180,E1 11709.383,E2 11709.383} C_VEL
LIN {X 0,Y 369.893,Z 843.44,A -85,B 0,C 180,E1 11716.593,E2 11716.593} C_VEL
LIN {X 0,Y 369.55,Z 843.44,A -85,B 0,C 180,E1 11724.1,E2 11724.1} C_VEL
LIN {X 0,Y 369.545,Z 844.196,A -85,B 0,C 180,E1 11724.674,E2 11724.674} C_VEL
LIN {X 0,Y 372.028,Z 849.24,A -85,B 0,C 180,E1 11725.702,E2 11725.702} C_VEL
LIN {X 0,Y 374.857,Z 852.173,A -85,B 0,C 180,E1 11726.697,E2 11726.697} C_VEL
LIN {X 0,Y 389.464,Z 872.701,A -85,B 0,C 180,E1 11731.366,E2 11731.366} C_VEL
LIN {X 0,Y 406.474,Z 899.701,A -85,B 0,C 180,E1 11736.11,E2 11736.11} C_VEL
LIN {X 0,Y 420.994,Z 929.848,A -85,B 0,C 180,E1 11740.263,E2 11740.263} C_VEL
LIN {X 0,Y 423.367,Z 936.888,A -85,B 0,C 180,E1 11741.061,E2 11741.061} C_VEL
LIN {X 0,Y 415.833,Z 979.301,A -85,B 0,C 180,E1 11743.302,E2 11743.302} C_VEL
LIN {X 0,Y 406.849,Z 1019.44,A -85,B 0,C 180,E1 11746.45,E2 11746.45} C_VEL
LIN {X 0,Y 397.353,Z 1055.953,A -85,B 0,C 180,E1 11750.438,E2 11750.438} C_VEL
LIN {X 0,Y 388.177,Z 1088.982,A -85,B 0,C 180,E1 11755.352,E2 11755.352} C_VEL
LIN {X 0,Y 380.548,Z 1117.349,A -85,B 0,C 180,E1 11761.069,E2 11761.069} C_VEL
LIN {X 0,Y 375.398,Z 1139.515,A -85,B 0,C 180,E1 11767.12,E2 11767.12} C_VEL
LIN {X 0,Y 372.406,Z 1156.3,A -85,B 0,C 180,E1 11773.522,E2 11773.522} C_VEL
LIN {X 0,Y 371.14,Z 1166.669,A -85,B 0,C 180,E1 11779.458,E2 11779.458} C_VEL
LIN {X 0,Y 370.807,Z 1172.516,A -85,B 0,C 180,E1 11785.332,E2 11785.332} C_VEL
LIN {X 0,Y 370.851,Z 1173.928,A -85,B 0,C 180,E1 11790,E2 11790} C_VEL
LIN {X 0,Y 370.82,Z 1172.766,A -85,B 0,C 180,E1 11794.122,E2 11794.122} C_VEL
LIN {X 0,Y 368.334,Z 1171.438,A -85,B 0,C 180,E1 11796.109,E2 11796.109} C_VEL
LIN {X 0,Y 363.176,Z 1168.473,A -85,B 0,C 180,E1 11799.088,E2 11799.088} C_VEL
LIN {X 0,Y 363.126,Z 1168.108,A -85,B 0,C 180,E1 11799.432,E2 11799.432} C_VEL
LIN {X 0,Y 364.214,Z 1158.411,A -85,B 0,C 180,E1 11805.623,E2 11805.623} C_VEL
LIN {X 0,Y 366.793,Z 1143.972,A -85,B 0,C 180,E1 11811.732,E2 11811.732} C_VEL
LIN {X 0,Y 371.872,Z 1122.659,A -85,B 0,C 180,E1 11818.147,E2 11818.147} C_VEL
LIN {X 0,Y 379.05,Z 1096.788,A -85,B 0,C 180,E1 11823.873,E2 11823.873} C_VEL
LIN {X 0,Y 388.398,Z 1064.738,A -85,B 0,C 180,E1 11829.112,E2 11829.112} C_VEL
LIN {X 0,Y 398.395,Z 1028.981,A -85,B 0,C 180,E1 11833.397,E2 11833.397} C_VEL
LIN {X 0,Y 408.085,Z 989.637,A -85,B 0,C 180,E1 11836.785,E2 11836.785} C_VEL
LIN {X 0,Y 416.364,Z 948.055,A -85,B 0,C 180,E1 11839.248,E2 11839.248} C_VEL
LIN {X 0,Y 417.455,Z 938.544,A -85,B 0,C 180,E1 11839.747,E2 11839.747} C_VEL
LIN {X 0,Y 404.14,Z 908.658,A -85,B 0,C 180,E1 11843.897,E2 11843.897} C_VEL
LIN {X 0,Y 388.188,Z 881.898,A -85,B 0,C 180,E1 11848.595,E2 11848.595} C_VEL
LIN {X 0,Y 375.374,Z 863.555,A -85,B 0,C 180,E1 11852.723,E2 11852.723} C_VEL
LIN {X 0,Y 370.263,Z 856.788,A -85,B 0,C 180,E1 11854.577,E2 11854.577} C_VEL
LIN {X 0,Y 365.684,Z 850.348,A -85,B 0,C 180,E1 11856.418,E2 11856.418} C_VEL
LIN {X 0,Y 362.086,Z 845.85,A -85,B 0,C 180,E1 11857.971,E2 11857.971} C_VEL
LIN {X 0,Y 361.77,Z 843.44,A -85,B 0,C 180,E1 11858.312,E2 11858.312} C_VEL
LIN {X 0,Y 362.003,Z 843.44,A -85,B 0,C 180,E1 11865.516,E2 11865.516} C_VEL
LIN {X 0,Y 362.472,Z 843.44,A -85,B 0,C 180,E1 11872.825,E2 11872.825} C_VEL
LIN {X 0,Y 362.849,Z 843.44,A -85,B 0,C 180,E1 11880,E2 11880} C_VEL
LIN {X 0,Y 362.476,Z 843.44,A -85,B 0,C 180,E1 11887.174,E2 11887.174} C_VEL
LIN {X 0,Y 362.134,Z 843.44,A -85,B 0,C 180,E1 11894.478,E2 11894.478} C_VEL
LIN {X 0,Y 361.701,Z 843.44,A -85,B 0,C 180,E1 11902.201,E2 11902.201} C_VEL
LIN {X 0,Y 363.372,Z 848.401,A -85,B 0,C 180,E1 11903.129,E2 11903.129} C_VEL
LIN {X 0,Y 367.175,Z 852.157,A -85,B 0,C 180,E1 11904.67,E2 11904.67} C_VEL
LIN {X 0,Y 377.95,Z 867.223,A -85,B 0,C 180,E1 11908.702,E2 11908.702} C_VEL
LIN {X 0,Y 392.176,Z 888.934,A -85,B 0,C 180,E1 11913.414,E2 11913.414} C_VEL
LIN {X 0,Y 406.748,Z 918.214,A -85,B 0,C 180,E1 11918.334,E2 11918.334} C_VEL
LIN {X 0,Y 414.908,Z 940.022,A -85,B 0,C 180,E1 11921.478,E2 11921.478} C_VEL
LIN {X 0,Y 407.066,Z 977.838,A -85,B 0,C 180,E1 11924.05,E2 11924.05} C_VEL
LIN {X 0,Y 397.835,Z 1013.339,A -85,B 0,C 180,E1 11927.375,E2 11927.375} C_VEL
LIN {X 0,Y 388.424,Z 1046.007,A -85,B 0,C 180,E1 11931.567,E2 11931.567} C_VEL
LIN {X 0,Y 379.301,Z 1075.513,A -85,B 0,C 180,E1 11936.66,E2 11936.66} C_VEL
LIN {X 0,Y 371.982,Z 1100.435,A -85,B 0,C 180,E1 11942.519,E2 11942.519} C_VEL
LIN {X 0,Y 366.853,Z 1120.16,A -85,B 0,C 180,E1 11948.904,E2 11948.904} C_VEL
LIN {X 0,Y 364.191,Z 1134.396,A -85,B 0,C 180,E1 11955.605,E2 11955.605} C_VEL
LIN {X 0,Y 363.097,Z 1142.324,A -85,B 0,C 180,E1 11961.636,E2 11961.636} C_VEL
LIN {X 0,Y 362.911,Z 1146.094,A -85,B 0,C 180,E1 11967.617,E2 11967.617} C_VEL
LIN {X 0,Y 362.926,Z 1145.5,A -85,B 0,C 180,E1 11973.755,E2 11973.755} C_VEL
LIN {X 0,Y 363.238,Z 1141.054,A -85,B 0,C 180,E1 11979.565,E2 11979.565} C_VEL
LIN {X 0,Y 364.72,Z 1130.9,A -85,B 0,C 180,E1 11986.217,E2 11986.217} C_VEL
LIN {X 0,Y 368.122,Z 1114.762,A -85,B 0,C 180,E1 11992.972,E2 11992.972} C_VEL
LIN {X 0,Y 374.037,Z 1093.205,A -85,B 0,C 180,E1 11999.278,E2 11999.278} C_VEL
LIN {X 0,Y 382.048,Z 1066.651,A -85,B 0,C 180,E1 12004.94,E2 12004.94} C_VEL
LIN {X 0,Y 391.338,Z 1036.144,A -85,B 0,C 180,E1 12009.738,E2 12009.738} C_VEL
LIN {X 0,Y 400.768,Z 1002.885,A -85,B 0,C 180,E1 12013.609,E2 12013.609} C_VEL
LIN {X 0,Y 409.374,Z 967.867,A -85,B 0,C 180,E1 12016.617,E2 12016.617} C_VEL
LIN {X 0,Y 414.551,Z 939.223,A -85,B 0,C 180,E1 12018.546,E2 12018.546} C_VEL
LIN {X 0,Y 403.588,Z 911.33,A -85,B 0,C 180,E1 12022.644,E2 12022.644} C_VEL
LIN {X 0,Y 389.48,Z 884.879,A -85,B 0,C 180,E1 12027.318,E2 12027.318} C_VEL
LIN {X 0,Y 375.662,Z 863.909,A -85,B 0,C 180,E1 12031.981,E2 12031.981} C_VEL
LIN {X 0,Y 370.328,Z 856.868,A -85,B 0,C 180,E1 12033.935,E2 12033.935} C_VEL
LIN {X 0,Y 365.662,Z 850.294,A -85,B 0,C 180,E1 12035.804,E2 12035.804} C_VEL
LIN {X 0,Y 362.004,Z 845.781,A -85,B 0,C 180,E1 12037.375,E2 12037.375} C_VEL
LIN {X 0,Y 361.671,Z 843.44,A -85,B 0,C 180,E1 12037.649,E2 12037.649} C_VEL
LIN {X 0,Y 362.094,Z 843.44,A -85,B 0,C 180,E1 12043.438,E2 12043.438} C_VEL
LIN {X 0,Y 362.34,Z 843.44,A -85,B 0,C 180,E1 12050.411,E2 12050.411} C_VEL
LIN {X 0,Y 362.757,Z 843.44,A -85,B 0,C 180,E1 12057.616,E2 12057.616} C_VEL
LIN {X 0,Y 362.709,Z 843.44,A -85,B 0,C 180,E1 12063.146,E2 12063.146} C_VEL
LIN {X 0,Y 362.307,Z 843.44,A -85,B 0,C 180,E1 12069.59,E2 12069.59} C_VEL
LIN {X 0,Y 361.953,Z 843.44,A -85,B 0,C 180,E1 12076.967,E2 12076.967} C_VEL
LIN {X 0,Y 361.757,Z 844.062,A -85,B 0,C 180,E1 12081.869,E2 12081.869} C_VEL
LIN {X 0,Y 363.938,Z 849.029,A -85,B 0,C 180,E1 12082.942,E2 12082.942} C_VEL
LIN {X 0,Y 367.065,Z 851.867,A -85,B 0,C 180,E1 12084.186,E2 12084.186} C_VEL
LIN {X 0,Y 371.256,Z 857.558,A -85,B 0,C 180,E1 12085.817,E2 12085.817} C_VEL
LIN {X 0,Y 386.625,Z 879.616,A -85,B 0,C 180,E1 12090.96,E2 12090.96} C_VEL
LIN {X 0,Y 402.866,Z 906.288,A -85,B 0,C 180,E1 12095.738,E2 12095.738} C_VEL
LIN {X 0,Y 416.707,Z 936.506,A -85,B 0,C 180,E1 12099.999,E2 12099.999} C_VEL
LIN {X 0,Y 417.468,Z 940.818,A -85,B 0,C 180,E1 12100.425,E2 12100.425} C_VEL
LIN {X 0,Y 409.955,Z 980.659,A -85,B 0,C 180,E1 12102.593,E2 12102.593} C_VEL
LIN {X 0,Y 400.764,Z 1019.952,A -85,B 0,C 180,E1 12105.728,E2 12105.728} C_VEL
LIN {X 0,Y 391.012,Z 1055.686,A -85,B 0,C 180,E1 12109.674,E2 12109.674} C_VEL
LIN {X 0,Y 381.288,Z 1089.044,A -85,B 0,C 180,E1 12114.713,E2 12114.713} C_VEL
LIN {X 0,Y 373.305,Z 1117.036,A -85,B 0,C 180,E1 12120.453,E2 12120.453} C_VEL
LIN {X 0,Y 367.643,Z 1139.974,A -85,B 0,C 180,E1 12126.886,E2 12126.886} C_VEL
LIN {X 0,Y 364.6,Z 1155.995,A -85,B 0,C 180,E1 12133.159,E2 12133.159} C_VEL
LIN {X 0,Y 363.277,Z 1166.369,A -85,B 0,C 180,E1 12139.227,E2 12139.227} C_VEL
LIN {X 0,Y 362.93,Z 1172.22,A -85,B 0,C 180,E1 12145.23,E2 12145.23} C_VEL
LIN {X 0,Y 362.955,Z 1173.632,A -85,B 0,C 180,E1 12150,E2 12150} C_VEL
LIN {X 0,Y 362.956,Z 1172.221,A -85,B 0,C 180,E1 12154.77,E2 12154.77} C_VEL
LIN {X 0,Y 363.126,Z 1168.108,A -85,B 0,C 180,E1 12159.432,E2 12159.432} C_VEL
LIN {X 0,Y 360.882,Z 1165.708,A -85,B 0,C 180,E1 12161.445,E2 12161.445} C_VEL
LIN {X 0,Y 356.11,Z 1160.991,A -85,B 0,C 180,E1 12164.443,E2 12164.443} C_VEL
LIN {X 0,Y 356.097,Z 1160.359,A -85,B 0,C 180,E1 12164.783,E2 12164.783} C_VEL
LIN {X 0,Y 358.811,Z 1145.4,A -85,B 0,C 180,E1 12171.592,E2 12171.592} C_VEL
LIN {X 0,Y 364.266,Z 1123.571,A -85,B 0,C 180,E1 12178.451,E2 12178.451} C_VEL
LIN {X 0,Y 372.216,Z 1096.48,A -85,B 0,C 180,E1 12184.582,E2 12184.582} C_VEL
LIN {X 0,Y 382.093,Z 1064.196,A -85,B 0,C 180,E1 12189.926,E2 12189.926} C_VEL
LIN {X 0,Y 392.657,Z 1028.023,A -85,B 0,C 180,E1 12194.283,E2 12194.283} C_VEL
LIN {X 0,Y 402.555,Z 989.494,A -85,B 0,C 180,E1 12197.613,E2 12197.613} C_VEL
LIN {X 0,Y 411.189,Z 947.592,A -85,B 0,C 180,E1 12200.104,E2 12200.104} C_VEL
LIN {X 0,Y 411.703,Z 941.744,A -85,B 0,C 180,E1 12200.444,E2 12200.444} C_VEL
LIN {X 0,Y 399.131,Z 912.913,A -85,B 0,C 180,E1 12204.626,E2 12204.626} C_VEL
LIN {X 0,Y 383.967,Z 886.76,A -85,B 0,C 180,E1 12209.423,E2 12209.423} C_VEL
LIN {X 0,Y 371.548,Z 868.853,A -85,B 0,C 180,E1 12213.652,E2 12213.652} C_VEL
LIN {X 0,Y 366.868,Z 862.693,A -85,B 0,C 180,E1 12215.432,E2 12215.432} C_VEL
LIN {X 0,Y 363.44,Z 857.542,A -85,B 0,C 180,E1 12216.878,E2 12216.878} C_VEL
LIN {X 0,Y 359.579,Z 852.087,A -85,B 0,C 180,E1 12218.634,E2 12218.634} C_VEL
LIN {X 0,Y 354.163,Z 845.542,A -85,B 0,C 180,E1 12221.364,E2 12221.364} C_VEL
LIN {X 0,Y 353.897,Z 843.44,A -85,B 0,C 180,E1 12221.672,E2 12221.672} C_VEL
LIN {X 0,Y 354.215,Z 843.44,A -85,B 0,C 180,E1 12228.476,E2 12228.476} C_VEL
LIN {X 0,Y 354.684,Z 843.44,A -85,B 0,C 180,E1 12235.119,E2 12235.119} C_VEL
LIN {X 0,Y 354.952,Z 843.44,A -85,B 0,C 180,E1 12240,E2 12240} C_VEL
LIN {X 0,Y 354.542,Z 843.44,A -85,B 0,C 180,E1 12247.335,E2 12247.335} C_VEL
LIN {X 0,Y 354.199,Z 843.44,A -85,B 0,C 180,E1 12254.81,E2 12254.81} C_VEL
LIN {X 0,Y 353.93,Z 843.641,A -85,B 0,C 180,E1 12258.89,E2 12258.89} C_VEL
LIN {X 0,Y 355.897,Z 848.75,A -85,B 0,C 180,E1 12260.106,E2 12260.106} C_VEL
LIN {X 0,Y 359.506,Z 852.022,A -85,B 0,C 180,E1 12261.816,E2 12261.816} C_VEL
LIN {X 0,Y 363.538,Z 857.606,A -85,B 0,C 180,E1 12263.643,E2 12263.643} C_VEL
LIN {X 0,Y 374.605,Z 872.898,A -85,B 0,C 180,E1 12268.015,E2 12268.015} C_VEL
LIN {X 0,Y 388.738,Z 895.898,A -85,B 0,C 180,E1 12273.083,E2 12273.083} C_VEL
LIN {X 0,Y 402.159,Z 924.027,A -85,B 0,C 180,E1 12277.942,E2 12277.942} C_VEL
LIN {X 0,Y 409.128,Z 943.963,A -85,B 0,C 180,E1 12280.867,E2 12280.867} C_VEL
LIN {X 0,Y 400.139,Z 984.063,A -85,B 0,C 180,E1 12283.711,E2 12283.711} C_VEL
LIN {X 0,Y 389.947,Z 1020.734,A -85,B 0,C 180,E1 12287.383,E2 12287.383} C_VEL
LIN {X 0,Y 379.715,Z 1053.853,A -85,B 0,C 180,E1 12291.978,E2 12291.978} C_VEL
LIN {X 0,Y 370.248,Z 1083.052,A -85,B 0,C 180,E1 12297.507,E2 12297.507} C_VEL
LIN {X 0,Y 362.687,Z 1107.421,A -85,B 0,C 180,E1 12303.877,E2 12303.877} C_VEL
LIN {X 0,Y 358.012,Z 1126.11,A -85,B 0,C 180,E1 12310.832,E2 12310.832} C_VEL
LIN {X 0,Y 355.789,Z 1138.435,A -85,B 0,C 180,E1 12317.756,E2 12317.756} C_VEL
LIN {X 0,Y 355.121,Z 1143.773,A -85,B 0,C 180,E1 12322.676,E2 12322.676} C_VEL
LIN {X 0,Y 355.02,Z 1146.389,A -85,B 0,C 180,E1 12327.564,E2 12327.564} C_VEL
LIN {X 0,Y 355.102,Z 1146.363,A -85,B 0,C 180,E1 12332.435,E2 12332.435} C_VEL
LIN {X 0,Y 355.284,Z 1142.533,A -85,B 0,C 180,E1 12338.549,E2 12338.549} C_VEL
LIN {X 0,Y 356.439,Z 1134.537,A -85,B 0,C 180,E1 12344.715,E2 12344.715} C_VEL
LIN {X 0,Y 359.299,Z 1120.255,A -85,B 0,C 180,E1 12351.561,E2 12351.561} C_VEL
LIN {X 0,Y 365.146,Z 1099.356,A -85,B 0,C 180,E1 12358.376,E2 12358.376} C_VEL
LIN {X 0,Y 373.425,Z 1073.227,A -85,B 0,C 180,E1 12364.454,E2 12364.454} C_VEL
LIN {X 0,Y 383.04,Z 1043.317,A -85,B 0,C 180,E1 12369.551,E2 12369.551} C_VEL
LIN {X 0,Y 393.593,Z 1008.211,A -85,B 0,C 180,E1 12373.91,E2 12373.91} C_VEL
LIN {X 0,Y 403.228,Z 971.307,A -85,B 0,C 180,E1 12377.213,E2 12377.213} C_VEL
LIN {X 0,Y 409.032,Z 943.346,A -85,B 0,C 180,E1 12379.105,E2 12379.105} C_VEL
LIN {X 0,Y 398.34,Z 915.107,A -85,B 0,C 180,E1 12383.402,E2 12383.402} C_VEL
LIN {X 0,Y 384.769,Z 889.142,A -85,B 0,C 180,E1 12388.199,E2 12388.199} C_VEL
LIN {X 0,Y 372.201,Z 869.944,A -85,B 0,C 180,E1 12392.714,E2 12392.714} C_VEL
LIN {X 0,Y 363.224,Z 857.412,A -85,B 0,C 180,E1 12396.336,E2 12396.336} C_VEL
LIN {X 0,Y 359.385,Z 851.667,A -85,B 0,C 180,E1 12398.099,E2 12398.099} C_VEL
LIN {X 0,Y 354.528,Z 846.28,A -85,B 0,C 180,E1 12400.498,E2 12400.498} C_VEL
LIN {X 0,Y 353.952,Z 843.44,A -85,B 0,C 180,E1 12401.031,E2 12401.031} C_VEL
LIN {X 0,Y 354.371,Z 843.44,A -85,B 0,C 180,E1 12408.351,E2 12408.351} C_VEL
LIN {X 0,Y 354.705,Z 843.44,A -85,B 0,C 180,E1 12415.119,E2 12415.119} C_VEL
LIN {X 0,Y 354.941,Z 843.44,A -85,B 0,C 180,E1 12422.437,E2 12422.437} C_VEL
LIN {X 0,Y 354.372,Z 843.44,A -85,B 0,C 180,E1 12429.807,E2 12429.807} C_VEL
LIN {X 0,Y 353.984,Z 843.44,A -85,B 0,C 180,E1 12437.361,E2 12437.361} C_VEL
LIN {X 0,Y 353.909,Z 843.815,A -85,B 0,C 180,E1 12438.489,E2 12438.489} C_VEL
LIN {X 0,Y 355.852,Z 848.63,A -85,B 0,C 180,E1 12439.669,E2 12439.669} C_VEL
LIN {X 0,Y 359.476,Z 851.772,A -85,B 0,C 180,E1 12441.371,E2 12441.371} C_VEL
LIN {X 0,Y 363.328,Z 857.463,A -85,B 0,C 180,E1 12443.131,E2 12443.131} C_VEL
LIN {X 0,Y 374.904,Z 873.244,A -85,B 0,C 180,E1 12447.574,E2 12447.574} C_VEL
LIN {X 0,Y 390.031,Z 896.533,A -85,B 0,C 180,E1 12452.548,E2 12452.548} C_VEL
LIN {X 0,Y 404.161,Z 923.479,A -85,B 0,C 180,E1 12457.002,E2 12457.002} C_VEL
LIN {X 0,Y 411.833,Z 943.213,A -85,B 0,C 180,E1 12459.694,E2 12459.694} C_VEL
LIN {X 0,Y 404.13,Z 982.142,A -85,B 0,C 180,E1 12461.875,E2 12461.875} C_VEL
LIN {X 0,Y 394.909,Z 1019.901,A -85,B 0,C 180,E1 12464.93,E2 12464.93} C_VEL
LIN {X 0,Y 384.697,Z 1055.69,A -85,B 0,C 180,E1 12468.926,E2 12468.926} C_VEL
LIN {X 0,Y 374.532,Z 1088.718,A -85,B 0,C 180,E1 12473.976,E2 12473.976} C_VEL
LIN {X 0,Y 366.433,Z 1115.817,A -85,B 0,C 180,E1 12479.588,E2 12479.588} C_VEL
LIN {X 0,Y 360.426,Z 1138.195,A -85,B 0,C 180,E1 12485.87,E2 12485.87} C_VEL
LIN {X 0,Y 356.821,Z 1155.689,A -85,B 0,C 180,E1 12492.781,E2 12492.781} C_VEL
LIN {X 0,Y 355.43,Z 1166.07,A -85,B 0,C 180,E1 12498.986,E2 12498.986} C_VEL
LIN {X 0,Y 355.019,Z 1171.922,A -85,B 0,C 180,E1 12505.124,E2 12505.124} C_VEL
LIN {X 0,Y 355.076,Z 1173.336,A -85,B 0,C 180,E1 12510,E2 12510} C_VEL
LIN {X 0,Y 355.047,Z 1171.923,A -85,B 0,C 180,E1 12514.876,E2 12514.876} C_VEL
LIN {X 0,Y 355.426,Z 1166.069,A -85,B 0,C 180,E1 12521.015,E2 12521.015} C_VEL
LIN {X 0,Y 356.097,Z 1160.359,A -85,B 0,C 180,E1 12524.783,E2 12524.783} C_VEL
LIN {X 0,Y 352.953,Z 1155.454,A -85,B 0,C 180,E1 12527.454,E2 12527.454} C_VEL
LIN {X 0,Y 350.121,Z 1149.862,A -85,B 0,C 180,E1 12530.142,E2 12530.142} C_VEL
LIN {X 0,Y 354.928,Z 1130.298,A -85,B 0,C 180,E1 12537.079,E2 12537.079} C_VEL
LIN {X 0,Y 362.545,Z 1104.863,A -85,B 0,C 180,E1 12543.53,E2 12543.53} C_VEL
LIN {X 0,Y 372.441,Z 1074.378,A -85,B 0,C 180,E1 12549.155,E2 12549.155} C_VEL
LIN {X 0,Y 383.141,Z 1040.537,A -85,B 0,C 180,E1 12553.724,E2 12553.724} C_VEL
LIN {X 0,Y 393.244,Z 1004.858,A -85,B 0,C 180,E1 12557.25,E2 12557.25} C_VEL
LIN {X 0,Y 402.592,Z 965.351,A -85,B 0,C 180,E1 12560.013,E2 12560.013} C_VEL
LIN {X 0,Y 405.957,Z 944.969,A -85,B 0,C 180,E1 12561.17,E2 12561.17} C_VEL
LIN {X 0,Y 393.817,Z 916.302,A -85,B 0,C 180,E1 12565.503,E2 12565.503} C_VEL
LIN {X 0,Y 378.888,Z 890.061,A -85,B 0,C 180,E1 12570.554,E2 12570.554} C_VEL
LIN {X 0,Y 365.937,Z 871.191,A -85,B 0,C 180,E1 12575.358,E2 12575.358} C_VEL
LIN {X 0,Y 360.445,Z 864.014,A -85,B 0,C 180,E1 12577.675,E2 12577.675} C_VEL
LIN {X 0,Y 356.133,Z 857.808,A -85,B 0,C 180,E1 12579.755,E2 12579.755} C_VEL
LIN {X 0,Y 352.041,Z 852.155,A -85,B 0,C 180,E1 12581.976,E2 12581.976} C_VEL
LIN {X 0,Y 346.59,Z 845.978,A -85,B 0,C 180,E1 12585.422,E2 12585.422} C_VEL
LIN {X 0,Y 346.178,Z 843.44,A -85,B 0,C 180,E1 12586.129,E2 12586.129} C_VEL
LIN {X 0,Y 346.591,Z 843.44,A -85,B 0,C 180,E1 12592.495,E2 12592.495} C_VEL
LIN {X 0,Y 347.075,Z 843.44,A -85,B 0,C 180,E1 12600,E2 12600} C_VEL
LIN {X 0,Y 346.63,Z 843.44,A -85,B 0,C 180,E1 12607.504,E2 12607.504} C_VEL
LIN {X 0,Y 346.344,Z 844.033,A -85,B 0,C 180,E1 12614.75,E2 12614.75} C_VEL
LIN {X 0,Y 348.236,Z 848.793,A -85,B 0,C 180,E1 12616.26,E2 12616.26} C_VEL
LIN {X 0,Y 352.051,Z 852.093,A -85,B 0,C 180,E1 12618.508,E2 12618.508} C_VEL
LIN {X 0,Y 355.863,Z 857.687,A -85,B 0,C 180,E1 12620.604,E2 12620.604} C_VEL
LIN {X 0,Y 358.104,Z 860.78,A -85,B 0,C 180,E1 12621.716,E2 12621.716} C_VEL
LIN {X 0,Y 363.831,Z 868.725,A -85,B 0,C 180,E1 12624.356,E2 12624.356} C_VEL
LIN {X 0,Y 372.211,Z 880.715,A -85,B 0,C 180,E1 12627.789,E2 12627.789} C_VEL
LIN {X 0,Y 384.797,Z 901.689,A -85,B 0,C 180,E1 12632.545,E2 12632.545} C_VEL
LIN {X 0,Y 397.279,Z 929.131,A -85,B 0,C 180,E1 12637.424,E2 12637.424} C_VEL
LIN {X 0,Y 403.188,Z 947.849,A -85,B 0,C 180,E1 12640.235,E2 12640.235} C_VEL
LIN {X 0,Y 394.145,Z 986.129,A -85,B 0,C 180,E1 12643.026,E2 12643.026} C_VEL
LIN {X 0,Y 383.559,Z 1022.517,A -85,B 0,C 180,E1 12646.746,E2 12646.746} C_VEL
LIN {X 0,Y 372.725,Z 1055.915,A -85,B 0,C 180,E1 12651.503,E2 12651.503} C_VEL
LIN {X 0,Y 363.27,Z 1083.691,A -85,B 0,C 180,E1 12656.89,E2 12656.89} C_VEL
LIN {X 0,Y 355.326,Z 1108.014,A -85,B 0,C 180,E1 12663.398,E2 12663.398} C_VEL
LIN {X 0,Y 350.384,Z 1126.338,A -85,B 0,C 180,E1 12670.36,E2 12670.36} C_VEL
LIN {X 0,Y 347.988,Z 1138.734,A -85,B 0,C 180,E1 12677.477,E2 12677.477} C_VEL
LIN {X 0,Y 347.268,Z 1144.07,A -85,B 0,C 180,E1 12682.509,E2 12682.509} C_VEL
LIN {X 0,Y 347.107,Z 1146.888,A -85,B 0,C 180,E1 12689.036,E2 12689.036} C_VEL
LIN {X 0,Y 347.171,Z 1145.663,A -85,B 0,C 180,E1 12694.987,E2 12694.987} C_VEL
LIN {X 0,Y 347.736,Z 1140.143,A -85,B 0,C 180,E1 12701.261,E2 12701.261} C_VEL
LIN {X 0,Y 349.554,Z 1130.322,A -85,B 0,C 180,E1 12707.589,E2 12707.589} C_VEL
LIN {X 0,Y 353.865,Z 1113.295,A -85,B 0,C 180,E1 12714.74,E2 12714.74} C_VEL
LIN {X 0,Y 360.622,Z 1091.646,A -85,B 0,C 180,E1 12721.115,E2 12721.115} C_VEL
LIN {X 0,Y 369.789,Z 1064.537,A -85,B 0,C 180,E1 12726.905,E2 12726.905} C_VEL
LIN {X 0,Y 380.746,Z 1031.441,A -85,B 0,C 180,E1 12732.029,E2 12732.029} C_VEL
LIN {X 0,Y 391.671,Z 994.914,A -85,B 0,C 180,E1 12736.095,E2 12736.095} C_VEL
LIN {X 0,Y 401.354,Z 956.682,A -85,B 0,C 180,E1 12739.106,E2 12739.106} C_VEL
LIN {X 0,Y 403.195,Z 946.544,A -85,B 0,C 180,E1 12739.791,E2 12739.791} C_VEL
LIN {X 0,Y 393.42,Z 919.841,A -85,B 0,C 180,E1 12744.013,E2 12744.013} C_VEL
LIN {X 0,Y 380.702,Z 894.8,A -85,B 0,C 180,E1 12748.819,E2 12748.819} C_VEL
LIN {X 0,Y 368.86,Z 875.867,A -85,B 0,C 180,E1 12753.428,E2 12753.428} C_VEL
LIN {X 0,Y 360.634,Z 864.249,A -85,B 0,C 180,E1 12756.928,E2 12756.928} C_VEL
LIN {X 0,Y 355.865,Z 857.675,A -85,B 0,C 180,E1 12759.236,E2 12759.236} C_VEL
LIN {X 0,Y 352.157,Z 852.282,A -85,B 0,C 180,E1 12761.255,E2 12761.255} C_VEL
LIN {X 0,Y 349.356,Z 849.769,A -85,B 0,C 180,E1 12762.858,E2 12762.858} C_VEL
LIN {X 0,Y 346.496,Z 845.209,A -85,B 0,C 180,E1 12764.853,E2 12764.853} C_VEL
LIN {X 0,Y 346.341,Z 843.44,A -85,B 0,C 180,E1 12765.169,E2 12765.169} C_VEL
LIN {X 0,Y 346.627,Z 843.44,A -85,B 0,C 180,E1 12772.792,E2 12772.792} C_VEL
LIN {X 0,Y 347.076,Z 843.44,A -85,B 0,C 180,E1 12780.28,E2 12780.28} C_VEL
LIN {X 0,Y 346.676,Z 843.44,A -85,B 0,C 180,E1 12787.503,E2 12787.503} C_VEL
LIN {X 0,Y 346.221,Z 843.601,A -85,B 0,C 180,E1 12794.272,E2 12794.272} C_VEL
LIN {X 0,Y 348.126,Z 848.73,A -85,B 0,C 180,E1 12795.813,E2 12795.813} C_VEL
LIN {X 0,Y 352.034,Z 852.163,A -85,B 0,C 180,E1 12798.105,E2 12798.105} C_VEL
LIN {X 0,Y 356.163,Z 857.806,A -85,B 0,C 180,E1 12800.328,E2 12800.328} C_VEL
LIN {X 0,Y 363.735,Z 868.455,A -85,B 0,C 180,E1 12803.805,E2 12803.805} C_VEL
LIN {X 0,Y 372.818,Z 881.074,A -85,B 0,C 180,E1 12807.342,E2 12807.342} C_VEL
LIN {X 0,Y 386.468,Z 902.757,A -85,B 0,C 180,E1 12812.057,E2 12812.057} C_VEL
LIN {X 0,Y 399.652,Z 929.08,A -85,B 0,C 180,E1 12816.54,E2 12816.54} C_VEL
LIN {X 0,Y 406.062,Z 947.037,A -85,B 0,C 180,E1 12819.015,E2 12819.015} C_VEL
LIN {X 0,Y 397.052,Z 989.276,A -85,B 0,C 180,E1 12821.528,E2 12821.528} C_VEL
LIN {X 0,Y 386.673,Z 1028.278,A -85,B 0,C 180,E1 12824.934,E2 12824.934} C_VEL
LIN {X 0,Y 375.845,Z 1063.871,A -85,B 0,C 180,E1 12829.275,E2 12829.275} C_VEL
LIN {X 0,Y 365.45,Z 1096.155,A -85,B 0,C 180,E1 12834.684,E2 12834.684} C_VEL
LIN {X 0,Y 356.961,Z 1123.257,A -85,B 0,C 180,E1 12840.912,E2 12840.912} C_VEL
LIN {X 0,Y 351.216,Z 1145.094,A -85,B 0,C 180,E1 12847.917,E2 12847.917} C_VEL
LIN {X 0,Y 348.339,Z 1160.158,A -85,B 0,C 180,E1 12854.935,E2 12854.935} C_VEL
LIN {X 0,Y 347.268,Z 1168.622,A -85,B 0,C 180,E1 12861.252,E2 12861.252} C_VEL
LIN {X 0,Y 347.117,Z 1172.685,A -85,B 0,C 180,E1 12867.509,E2 12867.509} C_VEL
LIN {X 0,Y 347.262,Z 1172.69,A -85,B 0,C 180,E1 12872.491,E2 12872.491} C_VEL
LIN {X 0,Y 347.284,Z 1168.623,A -85,B 0,C 180,E1 12878.748,E2 12878.748} C_VEL
LIN {X 0,Y 348.266,Z 1160.155,A -85,B 0,C 180,E1 12885.069,E2 12885.069} C_VEL
LIN {X 0,Y 350.121,Z 1149.862,A -85,B 0,C 180,E1 12890.142,E2 12890.142} C_VEL
LIN {X 0,Y 347.703,Z 1143.779,A -85,B 0,C 180,E1 12892.815,E2 12892.815} C_VEL
LIN {X 0,Y 345.628,Z 1136.895,A -85,B 0,C 180,E1 12895.472,E2 12895.472} C_VEL
LIN {X 0,Y 352.508,Z 1114.343,A -85,B 0,C 180,E1 12901.989,E2 12901.989} C_VEL
LIN {X 0,Y 361.941,Z 1086.337,A -85,B 0,C 180,E1 12907.896,E2 12907.896} C_VEL
LIN {X 0,Y 373.198,Z 1052.912,A -85,B 0,C 180,E1 12913.027,E2 12913.027} C_VEL
LIN {X 0,Y 384.606,Z 1015.811,A -85,B 0,C 180,E1 12917.135,E2 12917.135} C_VEL
LIN {X 0,Y 394.864,Z 976.408,A -85,B 0,C 180,E1 12920.223,E2 12920.223} C_VEL
LIN {X 0,Y 400.508,Z 948.749,A -85,B 0,C 180,E1 12921.829,E2 12921.829} C_VEL
LIN {X 0,Y 388.455,Z 919.792,A -85,B 0,C 180,E1 12926.412,E2 12926.412} C_VEL
LIN {X 0,Y 374.59,Z 894.961,A -85,B 0,C 180,E1 12931.422,E2 12931.422} C_VEL
LIN {X 0,Y 363.288,Z 877.939,A -85,B 0,C 180,E1 12935.9,E2 12935.9} C_VEL
LIN {X 0,Y 353.952,Z 864.928,A -85,B 0,C 180,E1 12940.302,E2 12940.302} C_VEL
LIN {X 0,Y 348.973,Z 858.175,A -85,B 0,C 180,E1 12943.151,E2 12943.151} C_VEL
LIN {X 0,Y 344.914,Z 853.083,A -85,B 0,C 180,E1 12945.915,E2 12945.915} C_VEL
LIN {X 0,Y 344.026,Z 851.006,A -85,B 0,C 180,E1 12946.687,E2 12946.687} C_VEL
LIN {X 0,Y 339.077,Z 846.368,A -85,B 0,C 180,E1 12951.362,E2 12951.362} C_VEL
LIN {X 0,Y 338.678,Z 843.44,A -85,B 0,C 180,E1 12952.318,E2 12952.318} C_VEL
LIN {X 0,Y 339.172,Z 843.44,A -85,B 0,C 180,E1 12960,E2 12960} C_VEL
LIN {X 0,Y 338.639,Z 843.44,A -85,B 0,C 180,E1 12968.004,E2 12968.004} C_VEL
LIN {X 0,Y 340.524,Z 848.754,A -85,B 0,C 180,E1 12970.835,E2 12970.835} C_VEL
LIN {X 0,Y 344.693,Z 852.048,A -85,B 0,C 180,E1 12974.336,E2 12974.336} C_VEL
LIN {X 0,Y 347.829,Z 857.387,A -85,B 0,C 180,E1 12976.651,E2 12976.651} C_VEL
LIN {X 0,Y 350.405,Z 859.929,A -85,B 0,C 180,E1 12978.192,E2 12978.192} C_VEL
LIN {X 0,Y 356.328,Z 868.628,A -85,B 0,C 180,E1 12981.487,E2 12981.487} C_VEL
LIN {X 0,Y 364.783,Z 880.296,A -85,B 0,C 180,E1 12985.415,E2 12985.415} C_VEL
LIN {X 0,Y 378.24,Z 902.626,A -85,B 0,C 180,E1 12990.989,E2 12990.989} C_VEL
LIN {X 0,Y 390.448,Z 929.325,A -85,B 0,C 180,E1 12996.075,E2 12996.075} C_VEL
LIN {X 0,Y 397.544,Z 950.643,A -85,B 0,C 180,E1 12999.517,E2 12999.517} C_VEL
LIN {X 0,Y 388.386,Z 987.558,A -85,B 0,C 180,E1 13002.263,E2 13002.263} C_VEL
LIN {X 0,Y 377.813,Z 1022.508,A -85,B 0,C 180,E1 13005.867,E2 13005.867} C_VEL
LIN {X 0,Y 366.38,Z 1056.218,A -85,B 0,C 180,E1 13010.709,E2 13010.709} C_VEL
LIN {X 0,Y 356.359,Z 1084.253,A -85,B 0,C 180,E1 13016.235,E2 13016.235} C_VEL
LIN {X 0,Y 348.347,Z 1107.61,A -85,B 0,C 180,E1 13022.568,E2 13022.568} C_VEL
LIN {X 0,Y 342.994,Z 1125.536,A -85,B 0,C 180,E1 13029.392,E2 13029.392} C_VEL
LIN {X 0,Y 340.528,Z 1137.176,A -85,B 0,C 180,E1 13035.893,E2 13035.893} C_VEL
LIN {X 0,Y 339.384,Z 1144.367,A -85,B 0,C 180,E1 13042.334,E2 13042.334} C_VEL
LIN {X 0,Y 339.223,Z 1146.982,A -85,B 0,C 180,E1 13047.45,E2 13047.45} C_VEL
LIN {X 0,Y 339.316,Z 1146.956,A -85,B 0,C 180,E1 13052.549,E2 13052.549} C_VEL
LIN {X 0,Y 339.558,Z 1143.131,A -85,B 0,C 180,E1 13058.948,E2 13058.948} C_VEL
LIN {X 0,Y 340.892,Z 1135.143,A -85,B 0,C 180,E1 13065.402,E2 13065.402} C_VEL
LIN {X 0,Y 344.222,Z 1120.925,A -85,B 0,C 180,E1 13072.53,E2 13072.53} C_VEL
LIN {X 0,Y 350.883,Z 1099.973,A -85,B 0,C 180,E1 13079.641,E2 13079.641} C_VEL
LIN {X 0,Y 360.087,Z 1073.845,A -85,B 0,C 180,E1 13085.923,E2 13085.923} C_VEL
LIN {X 0,Y 370.843,Z 1043.478,A -85,B 0,C 180,E1 13091.21,E2 13091.21} C_VEL
LIN {X 0,Y 382.048,Z 1009.224,A -85,B 0,C 180,E1 13095.542,E2 13095.542} C_VEL
LIN {X 0,Y 392.632,Z 971.659,A -85,B 0,C 180,E1 13098.942,E2 13098.942} C_VEL
LIN {X 0,Y 397.465,Z 950.727,A -85,B 0,C 180,E1 13100.385,E2 13100.385} C_VEL
LIN {X 0,Y 389.01,Z 925.805,A -85,B 0,C 180,E1 13104.42,E2 13104.42} C_VEL
LIN {X 0,Y 377.047,Z 900.971,A -85,B 0,C 180,E1 13109.319,E2 13109.319} C_VEL
LIN {X 0,Y 364.071,Z 879.042,A -85,B 0,C 180,E1 13114.778,E2 13114.778} C_VEL
LIN {X 0,Y 353.856,Z 864.974,A -85,B 0,C 180,E1 13119.659,E2 13119.659} C_VEL
LIN {X 0,Y 350.066,Z 858.883,A -85,B 0,C 180,E1 13121.871,E2 13121.871} C_VEL
LIN {X 0,Y 345.14,Z 853.602,A -85,B 0,C 180,E1 13125.036,E2 13125.036} C_VEL
LIN {X 0,Y 343.952,Z 850.967,A -85,B 0,C 180,E1 13126.038,E2 13126.038} C_VEL
LIN {X 0,Y 339.104,Z 846.234,A -85,B 0,C 180,E1 13130.556,E2 13130.556} C_VEL
LIN {X 0,Y 338.616,Z 843.44,A -85,B 0,C 180,E1 13131.673,E2 13131.673} C_VEL
LIN {X 0,Y 339.047,Z 843.44,A -85,B 0,C 180,E1 13137.449,E2 13137.449} C_VEL
LIN {X 0,Y 339.124,Z 843.44,A -85,B 0,C 180,E1 13142.55,E2 13142.55} C_VEL
LIN {X 0,Y 338.682,Z 843.85,A -85,B 0,C 180,E1 13148.084,E2 13148.084} C_VEL
LIN {X 0,Y 340.382,Z 848.575,A -85,B 0,C 180,E1 13150.386,E2 13150.386} C_VEL
LIN {X 0,Y 344.636,Z 851.985,A -85,B 0,C 180,E1 13153.935,E2 13153.935} C_VEL
LIN {X 0,Y 347.81,Z 857.401,A -85,B 0,C 180,E1 13156.258,E2 13156.258} C_VEL
LIN {X 0,Y 350.296,Z 859.789,A -85,B 0,C 180,E1 13157.732,E2 13157.732} C_VEL
LIN {X 0,Y 356.166,Z 868.107,A -85,B 0,C 180,E1 13160.899,E2 13160.899} C_VEL
LIN {X 0,Y 365.271,Z 880.602,A -85,B 0,C 180,E1 13164.968,E2 13164.968} C_VEL
LIN {X 0,Y 379.324,Z 902.589,A -85,B 0,C 180,E1 13170.312,E2 13170.312} C_VEL
LIN {X 0,Y 392.736,Z 929.14,A -85,B 0,C 180,E1 13175.193,E2 13175.193} C_VEL
LIN {X 0,Y 400.421,Z 948.596,A -85,B 0,C 180,E1 13178.156,E2 13178.156} C_VEL
LIN {X 0,Y 391.254,Z 990.971,A -85,B 0,C 180,E1 13180.788,E2 13180.788} C_VEL
LIN {X 0,Y 380.048,Z 1030.976,A -85,B 0,C 180,E1 13184.381,E2 13184.381} C_VEL
LIN {X 0,Y 368.979,Z 1065.643,A -85,B 0,C 180,E1 13188.741,E2 13188.741} C_VEL
LIN {X 0,Y 358.089,Z 1097.777,A -85,B 0,C 180,E1 13194.316,E2 13194.316} C_VEL
LIN {X 0,Y 349.568,Z 1123.612,A -85,B 0,C 180,E1 13200.442,E2 13200.442} C_VEL
LIN {X 0,Y 343.804,Z 1144.198,A -85,B 0,C 180,E1 13207.175,E2 13207.175} C_VEL
LIN {X 0,Y 340.54,Z 1159.855,A -85,B 0,C 180,E1 13214.581,E2 13214.581} C_VEL
LIN {X 0,Y 339.376,Z 1168.323,A -85,B 0,C 180,E1 13221.047,E2 13221.047} C_VEL
LIN {X 0,Y 339.214,Z 1172.388,A -85,B 0,C 180,E1 13227.451,E2 13227.451} C_VEL
LIN {X 0,Y 339.354,Z 1172.394,A -85,B 0,C 180,E1 13232.549,E2 13232.549} C_VEL
LIN {X 0,Y 339.39,Z 1168.324,A -85,B 0,C 180,E1 13238.953,E2 13238.953} C_VEL
LIN {X 0,Y 340.46,Z 1159.853,A -85,B 0,C 180,E1 13245.423,E2 13245.423} C_VEL
LIN {X 0,Y 343.849,Z 1144.149,A -85,B 0,C 180,E1 13252.843,E2 13252.843} C_VEL
LIN {X 0,Y 345.628,Z 1136.895,A -85,B 0,C 180,E1 13255.472,E2 13255.472} C_VEL
LIN {X 0,Y 344.035,Z 1129.568,A -85,B 0,C 180,E1 13258.11,E2 13258.11} C_VEL
LIN {X 0,Y 342.941,Z 1121.594,A -85,B 0,C 180,E1 13260.714,E2 13260.714} C_VEL
LIN {X 0,Y 352.035,Z 1095.555,A -85,B 0,C 180,E1 13266.879,E2 13266.879} C_VEL
LIN {X 0,Y 363.474,Z 1063.429,A -85,B 0,C 180,E1 13272.401,E2 13272.401} C_VEL
LIN {X 0,Y 375.183,Z 1028.026,A -85,B 0,C 180,E1 13276.81,E2 13276.81} C_VEL
LIN {X 0,Y 386.465,Z 989.245,A -85,B 0,C 180,E1 13280.223,E2 13280.223} C_VEL
LIN {X 0,Y 394.868,Z 952.172,A -85,B 0,C 180,E1 13282.54,E2 13282.54} C_VEL
LIN {X 0,Y 383.145,Z 923.248,A -85,B 0,C 180,E1 13287.327,E2 13287.327} C_VEL
LIN {X 0,Y 369.22,Z 897.628,A -85,B 0,C 180,E1 13292.792,E2 13292.792} C_VEL
LIN {X 0,Y 356.97,Z 879.131,A -85,B 0,C 180,E1 13298.169,E2 13298.169} C_VEL
LIN {X 0,Y 351.277,Z 871.489,A -85,B 0,C 180,E1 13301.124,E2 13301.124} C_VEL
LIN {X 0,Y 347.279,Z 865.659,A -85,B 0,C 180,E1 13303.549,E2 13303.549} C_VEL
LIN {X 0,Y 343.262,Z 860.208,A -85,B 0,C 180,E1 13306.414,E2 13306.414} C_VEL
LIN {X 0,Y 341.656,Z 858.322,A -85,B 0,C 180,E1 13307.732,E2 13307.732} C_VEL
LIN {X 0,Y 337.579,Z 852.963,A -85,B 0,C 180,E1 13312.132,E2 13312.132} C_VEL
LIN {X 0,Y 337.161,Z 851.196,A -85,B 0,C 180,E1 13312.93,E2 13312.93} C_VEL
LIN {X 0,Y 334.986,Z 850.289,A -85,B 0,C 180,E1 13323.228,E2 13323.228} C_VEL
LIN {X 0,Y 337.379,Z 851.951,A -85,B 0,C 180,E1 13327.953,E2 13327.953} C_VEL
LIN {X 0,Y 340.356,Z 857.453,A -85,B 0,C 180,E1 13331.632,E2 13331.632} C_VEL
LIN {X 0,Y 343.192,Z 859.884,A -85,B 0,C 180,E1 13333.994,E2 13333.994} C_VEL
LIN {X 0,Y 346.955,Z 865.436,A -85,B 0,C 180,E1 13336.779,E2 13336.779} C_VEL
LIN {X 0,Y 348.996,Z 868.348,A -85,B 0,C 180,E1 13338.105,E2 13338.105} C_VEL
LIN {X 0,Y 354.767,Z 876.69,A -85,B 0,C 180,E1 13341.376,E2 13341.376} C_VEL
LIN {X 0,Y 363.061,Z 889.055,A -85,B 0,C 180,E1 13345.461,E2 13345.461} C_VEL
LIN {X 0,Y 374.633,Z 909.31,A -85,B 0,C 180,E1 13350.621,E2 13350.621} C_VEL
LIN {X 0,Y 386.266,Z 936.263,A -85,B 0,C 180,E1 13355.872,E2 13355.872} C_VEL
LIN {X 0,Y 391.593,Z 954.955,A -85,B 0,C 180,E1 13358.869,E2 13358.869} C_VEL
LIN {X 0,Y 381.608,Z 992.74,A -85,B 0,C 180,E1 13361.82,E2 13361.82} C_VEL
LIN {X 0,Y 370.886,Z 1026.218,A -85,B 0,C 180,E1 13365.438,E2 13365.438} C_VEL
LIN {X 0,Y 360.116,Z 1056.52,A -85,B 0,C 180,E1 13369.889,E2 13369.889} C_VEL
LIN {X 0,Y 349.676,Z 1084.388,A -85,B 0,C 180,E1 13375.451,E2 13375.451} C_VEL
LIN {X 0,Y 341.315,Z 1107.415,A -85,B 0,C 180,E1 13381.783,E2 13381.783} C_VEL
LIN {X 0,Y 335.426,Z 1125.839,A -85,B 0,C 180,E1 13388.905,E2 13388.905} C_VEL
LIN {X 0,Y 332.727,Z 1137.477,A -85,B 0,C 180,E1 13395.555,E2 13395.555} C_VEL
LIN {X 0,Y 331.526,Z 1144.664,A -85,B 0,C 180,E1 13402.151,E2 13402.151} C_VEL
LIN {X 0,Y 331.34,Z 1147.278,A -85,B 0,C 180,E1 13407.389,E2 13407.389} C_VEL
LIN {X 0,Y 331.443,Z 1147.252,A -85,B 0,C 180,E1 13412.609,E2 13412.609} C_VEL
LIN {X 0,Y 331.709,Z 1143.43,A -85,B 0,C 180,E1 13419.161,E2 13419.161} C_VEL
LIN {X 0,Y 333.148,Z 1135.446,A -85,B 0,C 180,E1 13425.77,E2 13425.77} C_VEL
LIN {X 0,Y 336.704,Z 1121.313,A -85,B 0,C 180,E1 13433.023,E2 13433.023} C_VEL
LIN {X 0,Y 343.798,Z 1100.282,A -85,B 0,C 180,E1 13440.315,E2 13440.315} C_VEL
LIN {X 0,Y 353.506,Z 1074.155,A -85,B 0,C 180,E1 13446.699,E2 13446.699} C_VEL
LIN {X 0,Y 364.715,Z 1043.95,A -85,B 0,C 180,E1 13452.027,E2 13452.027} C_VEL
LIN {X 0,Y 376.434,Z 1009.586,A -85,B 0,C 180,E1 13456.412,E2 13456.412} C_VEL
LIN {X 0,Y 387.619,Z 971.218,A -85,B 0,C 180,E1 13459.891,E2 13459.891} C_VEL
LIN {X 0,Y 391.585,Z 952.968,A -85,B 0,C 180,E1 13461.237,E2 13461.237} C_VEL
LIN {X 0,Y 383.401,Z 928.837,A -85,B 0,C 180,E1 13465.368,E2 13465.368} C_VEL
LIN {X 0,Y 371.862,Z 904.25,A -85,B 0,C 180,E1 13470.464,E2 13470.464} C_VEL
LIN {X 0,Y 360.329,Z 884.88,A -85,B 0,C 180,E1 13475.655,E2 13475.655} C_VEL
LIN {X 0,Y 351.531,Z 871.989,A -85,B 0,C 180,E1 13480.22,E2 13480.22} C_VEL
LIN {X 0,Y 346.994,Z 865.409,A -85,B 0,C 180,E1 13483.013,E2 13483.013} C_VEL
LIN {X 0,Y 343.221,Z 859.94,A -85,B 0,C 180,E1 13485.764,E2 13485.764} C_VEL
LIN {X 0,Y 337.574,Z 852.916,A -85,B 0,C 180,E1 13491.323,E2 13491.323} C_VEL
LIN {X 0,Y 337.009,Z 851.156,A -85,B 0,C 180,E1 13492.281,E2 13492.281} C_VEL
LIN {X 0,Y 334.825,Z 850.113,A -85,B 0,C 180,E1 13502.906,E2 13502.906} C_VEL
LIN {X 0,Y 337.418,Z 852.021,A -85,B 0,C 180,E1 13507.791,E2 13507.791} C_VEL
LIN {X 0,Y 340.428,Z 857.488,A -85,B 0,C 180,E1 13511.376,E2 13511.376} C_VEL
LIN {X 0,Y 343.138,Z 859.753,A -85,B 0,C 180,E1 13513.591,E2 13513.591} C_VEL
LIN {X 0,Y 346.728,Z 865.255,A -85,B 0,C 180,E1 13516.216,E2 13516.216} C_VEL
LIN {X 0,Y 348.987,Z 868.181,A -85,B 0,C 180,E1 13517.618,E2 13517.618} C_VEL
LIN {X 0,Y 354.432,Z 875.89,A -85,B 0,C 180,E1 13520.654,E2 13520.654} C_VEL
LIN {X 0,Y 363.025,Z 888.045,A -85,B 0,C 180,E1 13524.643,E2 13524.643} C_VEL
LIN {X 0,Y 375.82,Z 909.127,A -85,B 0,C 180,E1 13529.876,E2 13529.876} C_VEL
LIN {X 0,Y 388.26,Z 934.701,A -85,B 0,C 180,E1 13534.696,E2 13534.696} C_VEL
LIN {X 0,Y 394.77,Z 953.411,A -85,B 0,C 180,E1 13537.57,E2 13537.57} C_VEL
LIN {X 0,Y 385.355,Z 993.015,A -85,B 0,C 180,E1 13540.06,E2 13540.06} C_VEL
LIN {X 0,Y 373.958,Z 1031.94,A -85,B 0,C 180,E1 13543.629,E2 13543.629} C_VEL
LIN {X 0,Y 362.785,Z 1065.41,A -85,B 0,C 180,E1 13547.894,E2 13547.894} C_VEL
LIN {X 0,Y 351.528,Z 1097.025,A -85,B 0,C 180,E1 13553.431,E2 13553.431} C_VEL
LIN {X 0,Y 342.32,Z 1123.619,A -85,B 0,C 180,E1 13559.857,E2 13559.857} C_VEL
LIN {X 0,Y 336.103,Z 1144.37,A -85,B 0,C 180,E1 13566.821,E2 13566.821} C_VEL
LIN {X 0,Y 332.729,Z 1159.55,A -85,B 0,C 180,E1 13574.21,E2 13574.21} C_VEL
LIN {X 0,Y 331.503,Z 1168.023,A -85,B 0,C 180,E1 13580.833,E2 13580.833} C_VEL
LIN {X 0,Y 331.333,Z 1172.092,A -85,B 0,C 180,E1 13587.39,E2 13587.39} C_VEL
LIN {X 0,Y 331.471,Z 1172.098,A -85,B 0,C 180,E1 13592.61,E2 13592.61} C_VEL
LIN {X 0,Y 331.514,Z 1168.025,A -85,B 0,C 180,E1 13599.167,E2 13599.167} C_VEL
LIN {X 0,Y 332.656,Z 1159.549,A -85,B 0,C 180,E1 13605.794,E2 13605.794} C_VEL
LIN {X 0,Y 336.157,Z 1144.347,A -85,B 0,C 180,E1 13613.188,E2 13613.188} C_VEL
LIN {X 0,Y 342.294,Z 1123.622,A -85,B 0,C 180,E1 13620.148,E2 13620.148} C_VEL
LIN {X 0,Y 342.941,Z 1121.594,A -85,B 0,C 180,E1 13620.714,E2 13620.714} C_VEL
LIN {X 0,Y 342.353,Z 1113.129,A -85,B 0,C 180,E1 13623.281,E2 13623.281} C_VEL
LIN {X 0,Y 342.153,Z 1104.056,A -85,B 0,C 180,E1 13625.794,E2 13625.794} C_VEL
LIN {X 0,Y 353.355,Z 1074.177,A -85,B 0,C 180,E1 13631.571,E2 13631.571} C_VEL
LIN {X 0,Y 365.856,Z 1039.353,A -85,B 0,C 180,E1 13636.418,E2 13636.418} C_VEL
LIN {X 0,Y 377.652,Z 1002.244,A -85,B 0,C 180,E1 13640.107,E2 13640.107} C_VEL
LIN {X 0,Y 387.904,Z 963.184,A -85,B 0,C 180,E1 13642.812,E2 13642.812} C_VEL
LIN {X 0,Y 389.28,Z 955.581,A -85,B 0,C 180,E1 13643.273,E2 13643.273} C_VEL
LIN {X 0,Y 378.302,Z 927.734,A -85,B 0,C 180,E1 13648.096,E2 13648.096} C_VEL
LIN {X 0,Y 365.734,Z 903.647,A -85,B 0,C 180,E1 13653.423,E2 13653.423} C_VEL
LIN {X 0,Y 354.526,Z 886.006,A -85,B 0,C 180,E1 13658.708,E2 13658.708} C_VEL
LIN {X 0,Y 348.802,Z 878.11,A -85,B 0,C 180,E1 13661.823,E2 13661.823} C_VEL
LIN {X 0,Y 345.235,Z 872.87,A -85,B 0,C 180,E1 13664.136,E2 13664.136} C_VEL
LIN {X 0,Y 341.407,Z 866.655,A -85,B 0,C 180,E1 13667.141,E2 13667.141} C_VEL
LIN {X 0,Y 336.52,Z 861.19,A -85,B 0,C 180,E1 13672.178,E2 13672.178} C_VEL
LIN {X 0,Y 335.759,Z 858.922,A -85,B 0,C 180,E1 13673.549,E2 13673.549} C_VEL
LIN {X 0,Y 334.024,Z 858.135,A -85,B 0,C 180,E1 13683.237,E2 13683.237} C_VEL
LIN {X 0,Y 336.221,Z 859.93,A -85,B 0,C 180,E1 13687.738,E2 13687.738} C_VEL
LIN {X 0,Y 339.866,Z 865.693,A -85,B 0,C 180,E1 13692.119,E2 13692.119} C_VEL
LIN {X 0,Y 341.739,Z 867.82,A -85,B 0,C 180,E1 13693.76,E2 13693.76} C_VEL
LIN {X 0,Y 345.849,Z 873.355,A -85,B 0,C 180,E1 13696.835,E2 13696.835} C_VEL
LIN {X 0,Y 355.725,Z 888.677,A -85,B 0,C 180,E1 13702.772,E2 13702.772} C_VEL
LIN {X 0,Y 366.435,Z 907.062,A -85,B 0,C 180,E1 13708.104,E2 13708.104} C_VEL
LIN {X 0,Y 376.713,Z 928.978,A -85,B 0,C 180,E1 13712.983,E2 13712.983} C_VEL
LIN {X 0,Y 385.483,Z 954.529,A -85,B 0,C 180,E1 13717.641,E2 13717.641} C_VEL
LIN {X 0,Y 385.571,Z 959.65,A -85,B 0,C 180,E1 13718.234,E2 13718.234} C_VEL
LIN {X 0,Y 374.737,Z 998.226,A -85,B 0,C 180,E1 13721.39,E2 13721.39} C_VEL
LIN {X 0,Y 362.448,Z 1034.325,A -85,B 0,C 180,E1 13725.575,E2 13725.575} C_VEL
LIN {X 0,Y 350.494,Z 1065.661,A -85,B 0,C 180,E1 13730.634,E2 13730.634} C_VEL
LIN {X 0,Y 339.372,Z 1093.849,A -85,B 0,C 180,E1 13736.996,E2 13736.996} C_VEL
LIN {X 0,Y 331.45,Z 1114.952,A -85,B 0,C 180,E1 13743.647,E2 13743.647} C_VEL
LIN {X 0,Y 326.47,Z 1131.412,A -85,B 0,C 180,E1 13751.122,E2 13751.122} C_VEL
LIN {X 0,Y 324.288,Z 1140.944,A -85,B 0,C 180,E1 13757.728,E2 13757.728} C_VEL
LIN {X 0,Y 323.473,Z 1146.601,A -85,B 0,C 180,E1 13764.646,E2 13764.646} C_VEL
LIN {X 0,Y 323.513,Z 1147.888,A -85,B 0,C 180,E1 13770,E2 13770} C_VEL
LIN {X 0,Y 323.495,Z 1146.556,A -85,B 0,C 180,E1 13775.353,E2 13775.353} C_VEL
LIN {X 0,Y 324.297,Z 1140.832,A -85,B 0,C 180,E1 13782.279,E2 13782.279} C_VEL
LIN {X 0,Y 326.852,Z 1129.939,A -85,B 0,C 180,E1 13789.555,E2 13789.555} C_VEL
LIN {X 0,Y 331.62,Z 1114.705,A -85,B 0,C 180,E1 13796.338,E2 13796.338} C_VEL
LIN {X 0,Y 340.005,Z 1092.307,A -85,B 0,C 180,E1 13803.314,E2 13803.314} C_VEL
LIN {X 0,Y 350.827,Z 1064.661,A -85,B 0,C 180,E1 13809.455,E2 13809.455} C_VEL
LIN {X 0,Y 362.969,Z 1032.684,A -85,B 0,C 180,E1 13814.552,E2 13814.552} C_VEL
LIN {X 0,Y 375.074,Z 996.795,A -85,B 0,C 180,E1 13818.658,E2 13818.658} C_VEL
LIN {X 0,Y 386.044,Z 956.746,A -85,B 0,C 180,E1 13821.898,E2 13821.898} C_VEL
LIN {X 0,Y 377.834,Z 931.908,A -85,B 0,C 180,E1 13826.35,E2 13826.35} C_VEL
LIN {X 0,Y 367.286,Z 908.961,A -85,B 0,C 180,E1 13831.331,E2 13831.331} C_VEL
LIN {X 0,Y 357.269,Z 891.311,A -85,B 0,C 180,E1 13836.262,E2 13836.262} C_VEL
LIN {X 0,Y 349.182,Z 878.969,A -85,B 0,C 180,E1 13840.761,E2 13840.761} C_VEL
LIN {X 0,Y 345.166,Z 872.84,A -85,B 0,C 180,E1 13843.404,E2 13843.404} C_VEL
LIN {X 0,Y 341.425,Z 866.844,A -85,B 0,C 180,E1 13846.34,E2 13846.34} C_VEL
LIN {X 0,Y 336.414,Z 860.792,A -85,B 0,C 180,E1 13851.537,E2 13851.537} C_VEL
LIN {X 0,Y 335.601,Z 858.875,A -85,B 0,C 180,E1 13852.898,E2 13852.898} C_VEL
LIN {X 0,Y 333.863,Z 857.959,A -85,B 0,C 180,E1 13862.915,E2 13862.915} C_VEL
LIN {X 0,Y 336.214,Z 859.779,A -85,B 0,C 180,E1 13867.495,E2 13867.495} C_VEL
LIN {X 0,Y 339.6,Z 865.534,A -85,B 0,C 180,E1 13871.523,E2 13871.523} C_VEL
LIN {X 0,Y 341.725,Z 867.597,A -85,B 0,C 180,E1 13873.303,E2 13873.303} C_VEL
LIN {X 0,Y 346.044,Z 873.422,A -85,B 0,C 180,E1 13876.464,E2 13876.464} C_VEL
LIN {X 0,Y 355.968,Z 888.119,A -85,B 0,C 180,E1 13882.1,E2 13882.1} C_VEL
LIN {X 0,Y 367.687,Z 907.289,A -85,B 0,C 180,E1 13887.496,E2 13887.496} C_VEL
LIN {X 0,Y 380.354,Z 932.176,A -85,B 0,C 180,E1 13892.763,E2 13892.763} C_VEL
LIN {X 0,Y 389.222,Z 955.582,A -85,B 0,C 180,E1 13896.733,E2 13896.733} C_VEL
LIN {X 0,Y 379.398,Z 995.552,A -85,B 0,C 180,E1 13899.353,E2 13899.353} C_VEL
LIN {X 0,Y 367.923,Z 1032.904,A -85,B 0,C 180,E1 13902.851,E2 13902.851} C_VEL
LIN {X 0,Y 356.014,Z 1066.96,A -85,B 0,C 180,E1 13907.299,E2 13907.299} C_VEL
LIN {X 0,Y 344.904,Z 1096.764,A -85,B 0,C 180,E1 13912.623,E2 13912.623} C_VEL
LIN {X 0,Y 335.302,Z 1122.925,A -85,B 0,C 180,E1 13919.028,E2 13919.028} C_VEL
LIN {X 0,Y 328.495,Z 1144.253,A -85,B 0,C 180,E1 13926.339,E2 13926.339} C_VEL
LIN {X 0,Y 324.947,Z 1159.246,A -85,B 0,C 180,E1 13933.822,E2 13933.822} C_VEL
LIN {X 0,Y 323.622,Z 1167.723,A -85,B 0,C 180,E1 13940.608,E2 13940.608} C_VEL
LIN {X 0,Y 323.428,Z 1171.795,A -85,B 0,C 180,E1 13947.326,E2 13947.326} C_VEL
LIN {X 0,Y 323.561,Z 1171.801,A -85,B 0,C 180,E1 13952.673,E2 13952.673} C_VEL
LIN {X 0,Y 323.631,Z 1167.726,A -85,B 0,C 180,E1 13959.393,E2 13959.393} C_VEL
LIN {X 0,Y 324.89,Z 1159.247,A -85,B 0,C 180,E1 13966.182,E2 13966.182} C_VEL
LIN {X 0,Y 328.533,Z 1144.243,A -85,B 0,C 180,E1 13973.666,E2 13973.666} C_VEL
LIN {X 0,Y 335.4,Z 1122.595,A -85,B 0,C 180,E1 13981.069,E2 13981.069} C_VEL
LIN {X 0,Y 342.153,Z 1104.056,A -85,B 0,C 180,E1 13985.794,E2 13985.794} C_VEL
LIN {X 0,Y 342.472,Z 1094.475,A -85,B 0,C 180,E1 13988.253,E2 13988.253} C_VEL
LIN {X 0,Y 343.136,Z 1084.32,A -85,B 0,C 180,E1 13990.639,E2 13990.639} C_VEL
LIN {X 0,Y 355.953,Z 1051.015,A -85,B 0,C 180,E1 13995.86,E2 13995.86} C_VEL
LIN {X 0,Y 368.05,Z 1016.27,A -85,B 0,C 180,E1 13999.786,E2 13999.786} C_VEL
LIN {X 0,Y 379.817,Z 976.012,A -85,B 0,C 180,E1 14002.978,E2 14002.978} C_VEL
LIN {X 0,Y 383.697,Z 958.811,A -85,B 0,C 180,E1 14004.057,E2 14004.057} C_VEL
LIN {X 0,Y 373.323,Z 931.633,A -85,B 0,C 180,E1 14008.985,E2 14008.985} C_VEL
LIN {X 0,Y 361.348,Z 908.337,A -85,B 0,C 180,E1 14014.409,E2 14014.409} C_VEL
LIN {X 0,Y 351.494,Z 892.389,A -85,B 0,C 180,E1 14019.421,E2 14019.421} C_VEL
LIN {X 0,Y 344.115,Z 880.85,A -85,B 0,C 180,E1 14024.083,E2 14024.083} C_VEL
LIN {X 0,Y 339.97,Z 874.589,A -85,B 0,C 180,E1 14027.363,E2 14027.363} C_VEL
LIN {X 0,Y 335.147,Z 868.146,A -85,B 0,C 180,E1 14032.806,E2 14032.806} C_VEL
LIN {X 0,Y 334.4,Z 866.623,A -85,B 0,C 180,E1 14034.173,E2 14034.173} C_VEL
LIN {X 0,Y 333.051,Z 865.979,A -85,B 0,C 180,E1 14043.246,E2 14043.246} C_VEL
LIN {X 0,Y 335.013,Z 867.753,A -85,B 0,C 180,E1 14047.521,E2 14047.521} C_VEL
LIN {X 0,Y 338.748,Z 873.535,A -85,B 0,C 180,E1 14052.16,E2 14052.16} C_VEL
LIN {X 0,Y 340.325,Z 875.898,A -85,B 0,C 180,E1 14053.617,E2 14053.617} C_VEL
LIN {X 0,Y 345.1,Z 883.19,A -85,B 0,C 180,E1 14057.412,E2 14057.412} C_VEL
LIN {X 0,Y 352.891,Z 895.453,A -85,B 0,C 180,E1 14062.302,E2 14062.302} C_VEL
LIN {X 0,Y 362.914,Z 913.615,A -85,B 0,C 180,E1 14067.679,E2 14067.679} C_VEL
LIN {X 0,Y 372.739,Z 935.946,A -85,B 0,C 180,E1 14072.753,E2 14072.753} C_VEL
LIN {X 0,Y 380.44,Z 960.16,A -85,B 0,C 180,E1 14077.268,E2 14077.268} C_VEL
LIN {X 0,Y 368.917,Z 1000.143,A -85,B 0,C 180,E1 14080.619,E2 14080.619} C_VEL
LIN {X 0,Y 356.726,Z 1034.624,A -85,B 0,C 180,E1 14084.667,E2 14084.667} C_VEL
LIN {X 0,Y 344.415,Z 1065.632,A -85,B 0,C 180,E1 14089.719,E2 14089.719} C_VEL
LIN {X 0,Y 332.559,Z 1094.153,A -85,B 0,C 180,E1 14096.23,E2 14096.23} C_VEL
LIN {X 0,Y 324.148,Z 1115.257,A -85,B 0,C 180,E1 14103.006,E2 14103.006} C_VEL
LIN {X 0,Y 318.816,Z 1131.714,A -85,B 0,C 180,E1 14110.651,E2 14110.651} C_VEL
LIN {X 0,Y 316.466,Z 1141.243,A -85,B 0,C 180,E1 14117.42,E2 14117.42} C_VEL
LIN {X 0,Y 315.603,Z 1146.897,A -85,B 0,C 180,E1 14124.512,E2 14124.512} C_VEL
LIN {X 0,Y 315.634,Z 1148.184,A -85,B 0,C 180,E1 14130,E2 14130} C_VEL
LIN {X 0,Y 315.625,Z 1146.853,A -85,B 0,C 180,E1 14135.487,E2 14135.487} C_VEL
LIN {X 0,Y 316.476,Z 1141.134,A -85,B 0,C 180,E1 14142.587,E2 14142.587} C_VEL
LIN {X 0,Y 319.214,Z 1130.245,A -85,B 0,C 180,E1 14150.043,E2 14150.043} C_VEL
LIN {X 0,Y 324.303,Z 1115.014,A -85,B 0,C 180,E1 14156.98,E2 14156.98} C_VEL
LIN {X 0,Y 333.237,Z 1092.615,A -85,B 0,C 180,E1 14164.082,E2 14164.082} C_VEL
LIN {X 0,Y 344.61,Z 1064.965,A -85,B 0,C 180,E1 14170.312,E2 14170.312} C_VEL
LIN {X 0,Y 357.217,Z 1032.993,A -85,B 0,C 180,E1 14175.468,E2 14175.468} C_VEL
LIN {X 0,Y 369.933,Z 996.73,A -85,B 0,C 180,E1 14179.626,E2 14179.626} C_VEL
LIN {X 0,Y 380.34,Z 959.849,A -85,B 0,C 180,E1 14182.683,E2 14182.683} C_VEL
LIN {X 0,Y 372.258,Z 934.871,A -85,B 0,C 180,E1 14187.37,E2 14187.37} C_VEL
LIN {X 0,Y 361.355,Z 910.664,A -85,B 0,C 180,E1 14192.977,E2 14192.977} C_VEL
LIN {X 0,Y 351.256,Z 892.844,A -85,B 0,C 180,E1 14198.501,E2 14198.501} C_VEL
LIN {X 0,Y 343.317,Z 880.327,A -85,B 0,C 180,E1 14203.728,E2 14203.728} C_VEL
LIN {X 0,Y 338.788,Z 873.562,A -85,B 0,C 180,E1 14207.558,E2 14207.558} C_VEL
LIN {X 0,Y 334.974,Z 867.768,A -85,B 0,C 180,E1 14212.152,E2 14212.152} C_VEL
LIN {X 0,Y 332.668,Z 865.641,A -85,B 0,C 180,E1 14217.4,E2 14217.4} C_VEL
LIN {X 0,Y 334.95,Z 867.104,A -85,B 0,C 180,E1 14227.035,E2 14227.035} C_VEL
LIN {X 0,Y 338.288,Z 873.243,A -85,B 0,C 180,E1 14231.33,E2 14231.33} C_VEL
LIN {X 0,Y 340.177,Z 875.255,A -85,B 0,C 180,E1 14232.998,E2 14232.998} C_VEL
LIN {X 0,Y 345.844,Z 883.846,A -85,B 0,C 180,E1 14237.21,E2 14237.21} C_VEL
LIN {X 0,Y 353.317,Z 894.946,A -85,B 0,C 180,E1 14241.615,E2 14241.615} C_VEL
LIN {X 0,Y 364.832,Z 914.68,A -85,B 0,C 180,E1 14247.245,E2 14247.245} C_VEL
LIN {X 0,Y 376.561,Z 939.238,A -85,B 0,C 180,E1 14252.54,E2 14252.54} C_VEL
LIN {X 0,Y 383.6,Z 960.111,A -85,B 0,C 180,E1 14256.068,E2 14256.068} C_VEL
LIN {X 0,Y 372.83,Z 1000.486,A -85,B 0,C 180,E1 14258.819,E2 14258.819} C_VEL
LIN {X 0,Y 360.12,Z 1039.032,A -85,B 0,C 180,E1 14262.627,E2 14262.627} C_VEL
LIN {X 0,Y 347.248,Z 1073.813,A -85,B 0,C 180,E1 14267.528,E2 14267.528} C_VEL
LIN {X 0,Y 335.469,Z 1103.852,A -85,B 0,C 180,E1 14273.415,E2 14273.415} C_VEL
LIN {X 0,Y 325.614,Z 1129.775,A -85,B 0,C 180,E1 14280.502,E2 14280.502} C_VEL
LIN {X 0,Y 319.659,Z 1148.568,A -85,B 0,C 180,E1 14287.812,E2 14287.812} C_VEL
LIN {X 0,Y 316.802,Z 1160.959,A -85,B 0,C 180,E1 14294.813,E2 14294.813} C_VEL
LIN {X 0,Y 315.608,Z 1168.658,A -85,B 0,C 180,E1 14301.753,E2 14301.753} C_VEL
LIN {X 0,Y 315.539,Z 1171.499,A -85,B 0,C 180,E1 14307.259,E2 14307.259} C_VEL
LIN {X 0,Y 315.678,Z 1171.505,A -85,B 0,C 180,E1 14312.74,E2 14312.74} C_VEL
LIN {X 0,Y 315.77,Z 1167.427,A -85,B 0,C 180,E1 14319.629,E2 14319.629} C_VEL
LIN {X 0,Y 317.103,Z 1158.943,A -85,B 0,C 180,E1 14326.591,E2 14326.591} C_VEL
LIN {X 0,Y 321.056,Z 1143.705,A -85,B 0,C 180,E1 14334.359,E2 14334.359} C_VEL
LIN {X 0,Y 328.482,Z 1121.919,A -85,B 0,C 180,E1 14341.925,E2 14341.925} C_VEL
LIN {X 0,Y 338.915,Z 1094.938,A -85,B 0,C 180,E1 14348.561,E2 14348.561} C_VEL
LIN {X 0,Y 343.136,Z 1084.32,A -85,B 0,C 180,E1 14350.639,E2 14350.639} C_VEL
LIN {X 0,Y 344.174,Z 1073.663,A -85,B 0,C 180,E1 14352.964,E2 14352.964} C_VEL
LIN {X 0,Y 345.705,Z 1062.408,A -85,B 0,C 180,E1 14355.173,E2 14355.173} C_VEL
LIN {X 0,Y 358.891,Z 1027.169,A -85,B 0,C 180,E1 14359.65,E2 14359.65} C_VEL
LIN {X 0,Y 371.52,Z 987.835,A -85,B 0,C 180,E1 14363.143,E2 14363.143} C_VEL
LIN {X 0,Y 378.126,Z 962.094,A -85,B 0,C 180,E1 14364.866,E2 14364.866} C_VEL
LIN {X 0,Y 368.866,Z 936.989,A -85,B 0,C 180,E1 14369.585,E2 14369.585} C_VEL
LIN {X 0,Y 357.813,Z 914.241,A -85,B 0,C 180,E1 14375.057,E2 14375.057} C_VEL
LIN {X 0,Y 346.407,Z 894.731,A -85,B 0,C 180,E1 14381.508,E2 14381.508} C_VEL
LIN {X 0,Y 341.245,Z 887.397,A -85,B 0,C 180,E1 14385.106,E2 14385.106} C_VEL
LIN {X 0,Y 337.601,Z 881.444,A -85,B 0,C 180,E1 14388.396,E2 14388.396} C_VEL
LIN {X 0,Y 333.733,Z 875.446,A -85,B 0,C 180,E1 14393.265,E2 14393.265} C_VEL
LIN {X 0,Y 331.64,Z 873.49,A -85,B 0,C 180,E1 14398.696,E2 14398.696} C_VEL
LIN {X 0,Y 333.679,Z 875.364,A -85,B 0,C 180,E1 14407.225,E2 14407.225} C_VEL
LIN {X 0,Y 337.366,Z 881.322,A -85,B 0,C 180,E1 14412.102,E2 14412.102} C_VEL
LIN {X 0,Y 343.25,Z 891.018,A -85,B 0,C 180,E1 14417.261,E2 14417.261} C_VEL
LIN {X 0,Y 350.478,Z 903.178,A -85,B 0,C 180,E1 14422.131,E2 14422.131} C_VEL
LIN {X 0,Y 359.06,Z 919.331,A -85,B 0,C 180,E1 14427.054,E2 14427.054} C_VEL
LIN {X 0,Y 368.105,Z 941.267,A -85,B 0,C 180,E1 14432.201,E2 14432.201} C_VEL
LIN {X 0,Y 374.856,Z 963.892,A -85,B 0,C 180,E1 14436.578,E2 14436.578} C_VEL
LIN {X 0,Y 363.369,Z 1001.522,A -85,B 0,C 180,E1 14439.773,E2 14439.773} C_VEL
LIN {X 0,Y 350.66,Z 1035.957,A -85,B 0,C 180,E1 14443.878,E2 14443.878} C_VEL
LIN {X 0,Y 337.626,Z 1067.336,A -85,B 0,C 180,E1 14449.104,E2 14449.104} C_VEL
LIN {X 0,Y 325.792,Z 1094.458,A -85,B 0,C 180,E1 14455.431,E2 14455.431} C_VEL
LIN {X 0,Y 316.925,Z 1115.56,A -85,B 0,C 180,E1 14462.339,E2 14462.339} C_VEL
LIN {X 0,Y 311.183,Z 1132.017,A -85,B 0,C 180,E1 14470.156,E2 14470.156} C_VEL
LIN {X 0,Y 308.41,Z 1142.617,A -85,B 0,C 180,E1 14478.106,E2 14478.106} C_VEL
LIN {X 0,Y 307.704,Z 1147.194,A -85,B 0,C 180,E1 14484.371,E2 14484.371} C_VEL
LIN {X 0,Y 307.738,Z 1148.48,A -85,B 0,C 180,E1 14490,E2 14490} C_VEL
LIN {X 0,Y 307.727,Z 1147.15,A -85,B 0,C 180,E1 14495.628,E2 14495.628} C_VEL
LIN {X 0,Y 308.663,Z 1141.483,A -85,B 0,C 180,E1 14502.864,E2 14502.864} C_VEL
LIN {X 0,Y 311.271,Z 1131.844,A -85,B 0,C 180,E1 14509.837,E2 14509.837} C_VEL
LIN {X 0,Y 317.061,Z 1115.321,A -85,B 0,C 180,E1 14517.648,E2 14517.648} C_VEL
LIN {X 0,Y 326.473,Z 1092.925,A -85,B 0,C 180,E1 14524.889,E2 14524.889} C_VEL
LIN {X 0,Y 338.337,Z 1065.599,A -85,B 0,C 180,E1 14531.139,E2 14531.139} C_VEL
LIN {X 0,Y 351.378,Z 1033.937,A -85,B 0,C 180,E1 14536.319,E2 14536.319} C_VEL
LIN {X 0,Y 364.31,Z 998.517,A -85,B 0,C 180,E1 14540.447,E2 14540.447} C_VEL
LIN {X 0,Y 374.644,Z 963.051,A -85,B 0,C 180,E1 14543.467,E2 14543.467} C_VEL
LIN {X 0,Y 366.827,Z 937.914,A -85,B 0,C 180,E1 14548.403,E2 14548.403} C_VEL
LIN {X 0,Y 356.492,Z 914.58,A -85,B 0,C 180,E1 14554.17,E2 14554.17} C_VEL
LIN {X 0,Y 348.136,Z 899.363,A -85,B 0,C 180,E1 14559.131,E2 14559.131} C_VEL
LIN {X 0,Y 341.086,Z 887.589,A -85,B 0,C 180,E1 14564.196,E2 14564.196} C_VEL
LIN {X 0,Y 337.109,Z 881.123,A -85,B 0,C 180,E1 14567.888,E2 14567.888} C_VEL
LIN {X 0,Y 333.578,Z 875.145,A -85,B 0,C 180,E1 14572.568,E2 14572.568} C_VEL
LIN {X 0,Y 331.424,Z 873.328,A -85,B 0,C 180,E1 14581.305,E2 14581.305} C_VEL
LIN {X 0,Y 333.745,Z 875.525,A -85,B 0,C 180,E1 14587.061,E2 14587.061} C_VEL
LIN {X 0,Y 337.432,Z 881.299,A -85,B 0,C 180,E1 14591.609,E2 14591.609} C_VEL
LIN {X 0,Y 343.697,Z 891.1,A -85,B 0,C 180,E1 14596.828,E2 14596.828} C_VEL
LIN {X 0,Y 351.121,Z 902.737,A -85,B 0,C 180,E1 14601.426,E2 14601.426} C_VEL
LIN {X 0,Y 362.243,Z 922.742,A -85,B 0,C 180,E1 14607.223,E2 14607.223} C_VEL
LIN {X 0,Y 373.07,Z 947.329,A -85,B 0,C 180,E1 14612.494,E2 14612.494} C_VEL
LIN {X 0,Y 378.106,Z 963.365,A -85,B 0,C 180,E1 14615.294,E2 14615.294} C_VEL
LIN {X 0,Y 366.965,Z 1003.113,A -85,B 0,C 180,E1 14618.083,E2 14618.083} C_VEL
LIN {X 0,Y 353.424,Z 1042.058,A -85,B 0,C 180,E1 14622.059,E2 14622.059} C_VEL
LIN {X 0,Y 340.291,Z 1075.803,A -85,B 0,C 180,E1 14626.982,E2 14626.982} C_VEL
LIN {X 0,Y 328.279,Z 1104.997,A -85,B 0,C 180,E1 14632.892,E2 14632.892} C_VEL
LIN {X 0,Y 318.042,Z 1130.48,A -85,B 0,C 180,E1 14640.12,E2 14640.12} C_VEL
LIN {X 0,Y 311.629,Z 1149.738,A -85,B 0,C 180,E1 14647.959,E2 14647.959} C_VEL
LIN {X 0,Y 308.627,Z 1162.632,A -85,B 0,C 180,E1 14655.85,E2 14655.85} C_VEL
LIN {X 0,Y 307.721,Z 1168.359,A -85,B 0,C 180,E1 14661.541,E2 14661.541} C_VEL
LIN {X 0,Y 307.632,Z 1171.202,A -85,B 0,C 180,E1 14667.189,E2 14667.189} C_VEL
LIN {X 0,Y 307.767,Z 1171.208,A -85,B 0,C 180,E1 14672.811,E2 14672.811} C_VEL
LIN {X 0,Y 307.908,Z 1167.128,A -85,B 0,C 180,E1 14679.877,E2 14679.877} C_VEL
LIN {X 0,Y 309.343,Z 1158.64,A -85,B 0,C 180,E1 14687.019,E2 14687.019} C_VEL
LIN {X 0,Y 313.639,Z 1143.268,A -85,B 0,C 180,E1 14695.035,E2 14695.035} C_VEL
LIN {X 0,Y 321.104,Z 1122.56,A -85,B 0,C 180,E1 14702.418,E2 14702.418} C_VEL
LIN {X 0,Y 332.481,Z 1094.629,A -85,B 0,C 180,E1 14709.451,E2 14709.451} C_VEL
LIN {X 0,Y 345.705,Z 1062.408,A -85,B 0,C 180,E1 14715.173,E2 14715.173} C_VEL
LIN {X 0,Y 347.555,Z 1050.633,A -85,B 0,C 180,E1 14717.301,E2 14717.301} C_VEL
LIN {X 0,Y 349.411,Z 1038.381,A -85,B 0,C 180,E1 14719.342,E2 14719.342} C_VEL
LIN {X 0,Y 362.779,Z 1000.541,A -85,B 0,C 180,E1 14723.123,E2 14723.123} C_VEL
LIN {X 0,Y 372.6,Z 965.59,A -85,B 0,C 180,E1 14725.636,E2 14725.636} C_VEL
LIN {X 0,Y 363.888,Z 941.162,A -85,B 0,C 180,E1 14730.465,E2 14730.465} C_VEL
LIN {X 0,Y 353.75,Z 919.222,A -85,B 0,C 180,E1 14735.943,E2 14735.943} C_VEL
LIN {X 0,Y 343.714,Z 901.595,A -85,B 0,C 180,E1 14742.103,E2 14742.103} C_VEL
LIN {X 0,Y 338.944,Z 894.508,A -85,B 0,C 180,E1 14745.662,E2 14745.662} C_VEL
LIN {X 0,Y 335.701,Z 888.919,A -85,B 0,C 180,E1 14748.823,E2 14748.823} C_VEL
LIN {X 0,Y 332.32,Z 882.716,A -85,B 0,C 180,E1 14753.727,E2 14753.727} C_VEL
LIN {X 0,Y 330.574,Z 881.416,A -85,B 0,C 180,E1 14762.616,E2 14762.616} C_VEL
LIN {X 0,Y 332.208,Z 883.141,A -85,B 0,C 180,E1 14767.011,E2 14767.011} C_VEL
LIN {X 0,Y 335.899,Z 889.122,A -85,B 0,C 180,E1 14772.156,E2 14772.156} C_VEL
LIN {X 0,Y 341.394,Z 899.299,A -85,B 0,C 180,E1 14777.358,E2 14777.358} C_VEL
LIN {X 0,Y 349.985,Z 914.556,A -85,B 0,C 180,E1 14783.307,E2 14783.307} C_VEL
LIN {X 0,Y 359.201,Z 934.802,A -85,B 0,C 180,E1 14788.95,E2 14788.95} C_VEL
LIN {X 0,Y 367.373,Z 959.418,A -85,B 0,C 180,E1 14794.286,E2 14794.286} C_VEL
LIN {X 0,Y 369.197,Z 967.02,A -85,B 0,C 180,E1 14795.755,E2 14795.755} C_VEL
LIN {X 0,Y 357.502,Z 1003.931,A -85,B 0,C 180,E1 14799,E2 14799} C_VEL
LIN {X 0,Y 345.317,Z 1035.714,A -85,B 0,C 180,E1 14802.827,E2 14802.827} C_VEL
LIN {X 0,Y 331.828,Z 1067.032,A -85,B 0,C 180,E1 14808.063,E2 14808.063} C_VEL
LIN {X 0,Y 319.022,Z 1094.951,A -85,B 0,C 180,E1 14814.656,E2 14814.656} C_VEL
LIN {X 0,Y 309.654,Z 1116.096,A -85,B 0,C 180,E1 14821.733,E2 14821.733} C_VEL
LIN {X 0,Y 303.556,Z 1132.32,A -85,B 0,C 180,E1 14829.636,E2 14829.636} C_VEL
LIN {X 0,Y 300.809,Z 1142.046,A -85,B 0,C 180,E1 14836.953,E2 14836.953} C_VEL
LIN {X 0,Y 299.825,Z 1147.491,A -85,B 0,C 180,E1 14844.223,E2 14844.223} C_VEL
LIN {X 0,Y 299.859,Z 1148.775,A -85,B 0,C 180,E1 14850,E2 14850} C_VEL
LIN {X 0,Y 299.848,Z 1147.448,A -85,B 0,C 180,E1 14855.776,E2 14855.776} C_VEL
LIN {X 0,Y 300.818,Z 1141.948,A -85,B 0,C 180,E1 14863.046,E2 14863.046} C_VEL
LIN {X 0,Y 303.628,Z 1132.15,A -85,B 0,C 180,E1 14870.358,E2 14870.358} C_VEL
LIN {X 0,Y 309.852,Z 1115.704,A -85,B 0,C 180,E1 14878.317,E2 14878.317} C_VEL
LIN {X 0,Y 319.764,Z 1093.396,A -85,B 0,C 180,E1 14885.679,E2 14885.679} C_VEL
LIN {X 0,Y 332.07,Z 1066.346,A -85,B 0,C 180,E1 14891.978,E2 14891.978} C_VEL
LIN {X 0,Y 345.89,Z 1034.086,A -85,B 0,C 180,E1 14897.312,E2 14897.312} C_VEL
LIN {X 0,Y 359.646,Z 997.676,A -85,B 0,C 180,E1 14901.541,E2 14901.541} C_VEL
LIN {X 0,Y 369.207,Z 967.162,A -85,B 0,C 180,E1 14904.111,E2 14904.111} C_VEL
LIN {X 0,Y 362.28,Z 943.26,A -85,B 0,C 180,E1 14908.973,E2 14908.973} C_VEL
LIN {X 0,Y 352.488,Z 919.754,A -85,B 0,C 180,E1 14914.991,E2 14914.991} C_VEL
LIN {X 0,Y 343.07,Z 901.802,A -85,B 0,C 180,E1 14921.239,E2 14921.239} C_VEL
LIN {X 0,Y 338.423,Z 894.271,A -85,B 0,C 180,E1 14924.98,E2 14924.98} C_VEL
LIN {X 0,Y 335.309,Z 888.684,A -85,B 0,C 180,E1 14928.152,E2 14928.152} C_VEL
LIN {X 0,Y 332.078,Z 882.67,A -85,B 0,C 180,E1 14932.904,E2 14932.904} C_VEL
LIN {X 0,Y 330.276,Z 881.145,A -85,B 0,C 180,E1 14941.309,E2 14941.309} C_VEL
LIN {X 0,Y 332.365,Z 883.147,A -85,B 0,C 180,E1 14946.763,E2 14946.763} C_VEL
LIN {X 0,Y 336.056,Z 889.108,A -85,B 0,C 180,E1 14951.658,E2 14951.658} C_VEL
LIN {X 0,Y 342.162,Z 899.406,A -85,B 0,C 180,E1 14956.905,E2 14956.905} C_VEL
LIN {X 0,Y 350.958,Z 914.022,A -85,B 0,C 180,E1 14962.515,E2 14962.515} C_VEL
LIN {X 0,Y 361.137,Z 934.727,A -85,B 0,C 180,E1 14968.106,E2 14968.106} C_VEL
LIN {X 0,Y 370.255,Z 958.309,A -85,B 0,C 180,E1 14973.031,E2 14973.031} C_VEL
LIN {X 0,Y 372.536,Z 966.739,A -85,B 0,C 180,E1 14974.507,E2 14974.507} C_VEL
LIN {X 0,Y 361.423,Z 1004.553,A -85,B 0,C 180,E1 14977.228,E2 14977.228} C_VEL
LIN {X 0,Y 347.984,Z 1041.739,A -85,B 0,C 180,E1 14981.055,E2 14981.055} C_VEL
LIN {X 0,Y 334.147,Z 1075.851,A -85,B 0,C 180,E1 14986.082,E2 14986.082} C_VEL
LIN {X 0,Y 321.715,Z 1104.737,A -85,B 0,C 180,E1 14992.018,E2 14992.018} C_VEL
LIN {X 0,Y 310.924,Z 1130.17,A -85,B 0,C 180,E1 14999.363,E2 14999.363} C_VEL
LIN {X 0,Y 304.069,Z 1149.431,A -85,B 0,C 180,E1 15007.381,E2 15007.381} C_VEL
LIN {X 0,Y 300.799,Z 1162.328,A -85,B 0,C 180,E1 15015.473,E2 15015.473} C_VEL
LIN {X 0,Y 299.865,Z 1168.061,A -85,B 0,C 180,E1 15021.317,E2 15021.317} C_VEL
LIN {X 0,Y 299.729,Z 1170.905,A -85,B 0,C 180,E1 15027.114,E2 15027.114} C_VEL
LIN {X 0,Y 299.88,Z 1170.912,A -85,B 0,C 180,E1 15032.885,E2 15032.885} C_VEL
LIN {X 0,Y 300.035,Z 1166.829,A -85,B 0,C 180,E1 15040.139,E2 15040.139} C_VEL
LIN {X 0,Y 301.594,Z 1158.337,A -85,B 0,C 180,E1 15047.47,E2 15047.47} C_VEL
LIN {X 0,Y 306.092,Z 1143.251,A -85,B 0,C 180,E1 15055.555,E2 15055.555} C_VEL
LIN {X 0,Y 314.453,Z 1121.632,A -85,B 0,C 180,E1 15063.418,E2 15063.418} C_VEL
LIN {X 0,Y 326.169,Z 1094.323,A -85,B 0,C 180,E1 15070.369,E2 15070.369} C_VEL
LIN {X 0,Y 339.683,Z 1062.854,A -85,B 0,C 180,E1 15076.042,E2 15076.042} C_VEL
LIN {X 0,Y 349.411,Z 1038.381,A -85,B 0,C 180,E1 15079.342,E2 15079.342} C_VEL
LIN {X 0,Y 351.565,Z 1025.588,A -85,B 0,C 180,E1 15081.281,E2 15081.281} C_VEL
LIN {X 0,Y 353.89,Z 1012.295,A -85,B 0,C 180,E1 15083.087,E2 15083.087} C_VEL
LIN {X 0,Y 366.079,Z 974.143,A -85,B 0,C 180,E1 15086.055,E2 15086.055} C_VEL
LIN {X 0,Y 367.179,Z 969.444,A -85,B 0,C 180,E1 15086.378,E2 15086.378} C_VEL
LIN {X 0,Y 359.406,Z 946.172,A -85,B 0,C 180,E1 15091.157,E2 15091.157} C_VEL
LIN {X 0,Y 349.642,Z 924.535,A -85,B 0,C 180,E1 15096.824,E2 15096.824} C_VEL
LIN {X 0,Y 340.965,Z 908.486,A -85,B 0,C 180,E1 15102.619,E2 15102.619} C_VEL
LIN {X 0,Y 336.472,Z 901.424,A -85,B 0,C 180,E1 15106.299,E2 15106.299} C_VEL
LIN {X 0,Y 333.74,Z 896.347,A -85,B 0,C 180,E1 15109.251,E2 15109.251} C_VEL
LIN {X 0,Y 330.3,Z 889.835,A -85,B 0,C 180,E1 15114.757,E2 15114.757} C_VEL
LIN {X 0,Y 329.403,Z 889.487,A -85,B 0,C 180,E1 15123.94,E2 15123.94} C_VEL
LIN {X 0,Y 330.591,Z 891.042,A -85,B 0,C 180,E1 15126.881,E2 15126.881} C_VEL
LIN {X 0,Y 334.502,Z 898.364,A -85,B 0,C 180,E1 15132.704,E2 15132.704} C_VEL
LIN {X 0,Y 339.111,Z 906.849,A -85,B 0,C 180,E1 15137.145,E2 15137.145} C_VEL
LIN {X 0,Y 346.149,Z 920.049,A -85,B 0,C 180,E1 15142.457,E2 15142.457} C_VEL
LIN {X 0,Y 354.668,Z 939.88,A -85,B 0,C 180,E1 15148.25,E2 15148.25} C_VEL
LIN {X 0,Y 362.327,Z 964.721,A -85,B 0,C 180,E1 15153.822,E2 15153.822} C_VEL
LIN {X 0,Y 363.49,Z 971.586,A -85,B 0,C 180,E1 15155.079,E2 15155.079} C_VEL
LIN {X 0,Y 349.907,Z 1011.251,A -85,B 0,C 180,E1 15158.721,E2 15158.721} C_VEL
LIN {X 0,Y 335.77,Z 1045.501,A -85,B 0,C 180,E1 15163.242,E2 15163.242} C_VEL
LIN {X 0,Y 321.608,Z 1076.071,A -85,B 0,C 180,E1 15168.936,E2 15168.936} C_VEL
LIN {X 0,Y 308.811,Z 1102.693,A -85,B 0,C 180,E1 15176.039,E2 15176.039} C_VEL
LIN {X 0,Y 299.805,Z 1122.745,A -85,B 0,C 180,E1 15183.791,E2 15183.791} C_VEL
LIN {X 0,Y 294.554,Z 1137.103,A -85,B 0,C 180,E1 15192.098,E2 15192.098} C_VEL
LIN {X 0,Y 292.356,Z 1145.152,A -85,B 0,C 180,E1 15199.782,E2 15199.782} C_VEL
LIN {X 0,Y 291.845,Z 1148.76,A -85,B 0,C 180,E1 15207.036,E2 15207.036} C_VEL
LIN {X 0,Y 291.97,Z 1148.735,A -85,B 0,C 180,E1 15212.962,E2 15212.962} C_VEL
LIN {X 0,Y 292.393,Z 1145.07,A -85,B 0,C 180,E1 15220.222,E2 15220.222} C_VEL
LIN {X 0,Y 294.583,Z 1136.962,A -85,B 0,C 180,E1 15227.899,E2 15227.899} C_VEL
LIN {X 0,Y 299.897,Z 1122.551,A -85,B 0,C 180,E1 15236.201,E2 15236.201} C_VEL
LIN {X 0,Y 309.163,Z 1102.031,A -85,B 0,C 180,E1 15244.071,E2 15244.071} C_VEL
LIN {X 0,Y 321.771,Z 1075.697,A -85,B 0,C 180,E1 15251.038,E2 15251.038} C_VEL
LIN {X 0,Y 335.943,Z 1044.892,A -85,B 0,C 180,E1 15256.756,E2 15256.756} C_VEL
LIN {X 0,Y 350.254,Z 1010.148,A -85,B 0,C 180,E1 15261.294,E2 15261.294} C_VEL
LIN {X 0,Y 363.351,Z 972.183,A -85,B 0,C 180,E1 15264.754,E2 15264.754} C_VEL
LIN {X 0,Y 361.447,Z 961.237,A -85,B 0,C 180,E1 15266.79,E2 15266.79} C_VEL
LIN {X 0,Y 353.941,Z 938.509,A -85,B 0,C 180,E1 15272.033,E2 15272.033} C_VEL
LIN {X 0,Y 345.469,Z 918.968,A -85,B 0,C 180,E1 15277.813,E2 15277.813} C_VEL
LIN {X 0,Y 337.372,Z 902.996,A -85,B 0,C 180,E1 15284.267,E2 15284.267} C_VEL
LIN {X 0,Y 333.224,Z 896.124,A -85,B 0,C 180,E1 15288.573,E2 15288.573} C_VEL
LIN {X 0,Y 329.971,Z 889.778,A -85,B 0,C 180,E1 15294.095,E2 15294.095} C_VEL
LIN {X 0,Y 329.07,Z 889.099,A -85,B 0,C 180,E1 15302.628,E2 15302.628} C_VEL
LIN {X 0,Y 330.744,Z 891.014,A -85,B 0,C 180,E1 15306.632,E2 15306.632} C_VEL
LIN {X 0,Y 335.079,Z 898.555,A -85,B 0,C 180,E1 15312.352,E2 15312.352} C_VEL
LIN {X 0,Y 341.736,Z 909.583,A -85,B 0,C 180,E1 15318.005,E2 15318.005} C_VEL
LIN {X 0,Y 351.533,Z 928.386,A -85,B 0,C 180,E1 15324.351,E2 15324.351} C_VEL
LIN {X 0,Y 361.365,Z 951.573,A -85,B 0,C 180,E1 15330.072,E2 15330.072} C_VEL
LIN {X 0,Y 367.084,Z 969.266,A -85,B 0,C 180,E1 15333.604,E2 15333.604} C_VEL
LIN {X 0,Y 355.291,Z 1007.933,A -85,B 0,C 180,E1 15336.521,E2 15336.521} C_VEL
LIN {X 0,Y 341.658,Z 1043.919,A -85,B 0,C 180,E1 15340.348,E2 15340.348} C_VEL
LIN {X 0,Y 328.314,Z 1075.469,A -85,B 0,C 180,E1 15345.074,E2 15345.074} C_VEL
LIN {X 0,Y 315.095,Z 1104.658,A -85,B 0,C 180,E1 15351.149,E2 15351.149} C_VEL
LIN {X 0,Y 303.868,Z 1129.859,A -85,B 0,C 180,E1 15358.572,E2 15358.572} C_VEL
LIN {X 0,Y 296.443,Z 1149.342,A -85,B 0,C 180,E1 15366.892,E2 15366.892} C_VEL
LIN {X 0,Y 292.979,Z 1162.025,A -85,B 0,C 180,E1 15375.077,E2 15375.077} C_VEL
LIN {X 0,Y 291.981,Z 1167.761,A -85,B 0,C 180,E1 15381.081,E2 15381.081} C_VEL
LIN {X 0,Y 291.82,Z 1170.608,A -85,B 0,C 180,E1 15387.036,E2 15387.036} C_VEL
LIN {X 0,Y 291.965,Z 1170.615,A -85,B 0,C 180,E1 15392.963,E2 15392.963} C_VEL
LIN {X 0,Y 292.246,Z 1165.892,A -85,B 0,C 180,E1 15401.178,E2 15401.178} C_VEL
LIN {X 0,Y 294.182,Z 1156.77,A -85,B 0,C 180,E1 15408.755,E2 15408.755} C_VEL
LIN {X 0,Y 298.675,Z 1142.943,A -85,B 0,C 180,E1 15416.237,E2 15416.237} C_VEL
LIN {X 0,Y 307.48,Z 1121.566,A -85,B 0,C 180,E1 15424.19,E2 15424.19} C_VEL
LIN {X 0,Y 319.922,Z 1094.016,A -85,B 0,C 180,E1 15431.327,E2 15431.327} C_VEL
LIN {X 0,Y 334.027,Z 1062.544,A -85,B 0,C 180,E1 15437.059,E2 15437.059} C_VEL
LIN {X 0,Y 348.573,Z 1026.689,A -85,B 0,C 180,E1 15441.668,E2 15441.668} C_VEL
LIN {X 0,Y 353.89,Z 1012.295,A -85,B 0,C 180,E1 15443.087,E2 15443.087} C_VEL
LIN {X 0,Y 356.132,Z 998.557,A -85,B 0,C 180,E1 15444.814,E2 15444.814} C_VEL
LIN {X 0,Y 357.854,Z 986.303,A -85,B 0,C 180,E1 15446.265,E2 15446.265} C_VEL
LIN {X 0,Y 358.372,Z 984.389,A -85,B 0,C 180,E1 15446.411,E2 15446.411} C_VEL
LIN {X 0,Y 361.774,Z 973.202,A -85,B 0,C 180,E1 15447.164,E2 15447.164} C_VEL
LIN {X 0,Y 354.416,Z 950.216,A -85,B 0,C 180,E1 15452.074,E2 15452.074} C_VEL
LIN {X 0,Y 345.444,Z 929.405,A -85,B 0,C 180,E1 15457.848,E2 15457.848} C_VEL
LIN {X 0,Y 337.719,Z 914.536,A -85,B 0,C 180,E1 15463.534,E2 15463.534} C_VEL
LIN {X 0,Y 331.99,Z 904.117,A -85,B 0,C 180,E1 15469.193,E2 15469.193} C_VEL
LIN {X 0,Y 328.778,Z 897.595,A -85,B 0,C 180,E1 15474.733,E2 15474.733} C_VEL
LIN {X 0,Y 327.807,Z 897.225,A -85,B 0,C 180,E1 15483.959,E2 15483.959} C_VEL
LIN {X 0,Y 328.795,Z 898.78,A -85,B 0,C 180,E1 15486.753,E2 15486.753} C_VEL
LIN {X 0,Y 332.341,Z 905.911,A -85,B 0,C 180,E1 15492.454,E2 15492.454} C_VEL
LIN {X 0,Y 336.625,Z 914.433,A -85,B 0,C 180,E1 15497.024,E2 15497.024} C_VEL
LIN {X 0,Y 343.704,Z 928.94,A -85,B 0,C 180,E1 15502.78,E2 15502.78} C_VEL
LIN {X 0,Y 351.108,Z 947.675,A -85,B 0,C 180,E1 15508.212,E2 15508.212} C_VEL
LIN {X 0,Y 357.594,Z 971.339,A -85,B 0,C 180,E1 15513.618,E2 15513.618} C_VEL
LIN {X 0,Y 358.081,Z 974.686,A -85,B 0,C 180,E1 15514.251,E2 15514.251} C_VEL
LIN {X 0,Y 344.167,Z 1013.391,A -85,B 0,C 180,E1 15517.887,E2 15517.887} C_VEL
LIN {X 0,Y 329.396,Z 1047.656,A -85,B 0,C 180,E1 15522.514,E2 15522.514} C_VEL
LIN {X 0,Y 314.776,Z 1077.85,A -85,B 0,C 180,E1 15528.305,E2 15528.305} C_VEL
LIN {X 0,Y 301.747,Z 1103.623,A -85,B 0,C 180,E1 15535.388,E2 15535.388} C_VEL
LIN {X 0,Y 292.425,Z 1123.195,A -85,B 0,C 180,E1 15543.158,E2 15543.158} C_VEL
LIN {X 0,Y 286.883,Z 1137.405,A -85,B 0,C 180,E1 15551.603,E2 15551.603} C_VEL
LIN {X 0,Y 284.498,Z 1145.597,A -85,B 0,C 180,E1 15559.692,E2 15559.692} C_VEL
LIN {X 0,Y 283.962,Z 1149.056,A -85,B 0,C 180,E1 15566.953,E2 15566.953} C_VEL
LIN {X 0,Y 284.073,Z 1149.031,A -85,B 0,C 180,E1 15573.045,E2 15573.045} C_VEL
LIN {X 0,Y 284.534,Z 1145.511,A -85,B 0,C 180,E1 15580.319,E2 15580.319} C_VEL
LIN {X 0,Y 286.919,Z 1137.266,A -85,B 0,C 180,E1 15588.394,E2 15588.394} C_VEL
LIN {X 0,Y 292.534,Z 1123.01,A -85,B 0,C 180,E1 15596.831,E2 15596.831} C_VEL
LIN {X 0,Y 302.783,Z 1101.725,A -85,B 0,C 180,E1 15605.119,E2 15605.119} C_VEL
LIN {X 0,Y 315.659,Z 1076.006,A -85,B 0,C 180,E1 15612.011,E2 15612.011} C_VEL
LIN {X 0,Y 330.248,Z 1045.679,A -85,B 0,C 180,E1 15617.704,E2 15617.704} C_VEL
LIN {X 0,Y 344.921,Z 1011.421,A -85,B 0,C 180,E1 15622.232,E2 15622.232} C_VEL
LIN {X 0,Y 358.164,Z 973.945,A -85,B 0,C 180,E1 15625.732,E2 15625.732} C_VEL
LIN {X 0,Y 351.856,Z 950.214,A -85,B 0,C 180,E1 15631.028,E2 15631.028} C_VEL
LIN {X 0,Y 344.07,Z 930.047,A -85,B 0,C 180,E1 15636.753,E2 15636.753} C_VEL
LIN {X 0,Y 336.872,Z 914.863,A -85,B 0,C 180,E1 15642.569,E2 15642.569} C_VEL
LIN {X 0,Y 333.043,Z 907.585,A -85,B 0,C 180,E1 15646.432,E2 15646.432} C_VEL
LIN {X 0,Y 331.1,Z 903.661,A -85,B 0,C 180,E1 15648.832,E2 15648.832} C_VEL
LIN {X 0,Y 328.348,Z 897.51,A -85,B 0,C 180,E1 15654.065,E2 15654.065} C_VEL
LIN {X 0,Y 327.552,Z 896.861,A -85,B 0,C 180,E1 15662.641,E2 15662.641} C_VEL
LIN {X 0,Y 329.028,Z 898.702,A -85,B 0,C 180,E1 15666.419,E2 15666.419} C_VEL
LIN {X 0,Y 332.979,Z 906.202,A -85,B 0,C 180,E1 15672.182,E2 15672.182} C_VEL
LIN {X 0,Y 339.09,Z 916.781,A -85,B 0,C 180,E1 15677.648,E2 15677.648} C_VEL
LIN {X 0,Y 347.616,Z 934.106,A -85,B 0,C 180,E1 15683.675,E2 15683.675} C_VEL
LIN {X 0,Y 356.243,Z 955.402,A -85,B 0,C 180,E1 15689.151,E2 15689.151} C_VEL
LIN {X 0,Y 361.713,Z 973.154,A -85,B 0,C 180,E1 15692.842,E2 15692.842} C_VEL
LIN {X 0,Y 348.887,Z 1012.171,A -85,B 0,C 180,E1 15695.862,E2 15695.862} C_VEL
LIN {X 0,Y 334.434,Z 1048.359,A -85,B 0,C 180,E1 15699.909,E2 15699.909} C_VEL
LIN {X 0,Y 319.962,Z 1080.516,A -85,B 0,C 180,E1 15705.025,E2 15705.025} C_VEL
LIN {X 0,Y 306.664,Z 1108.501,A -85,B 0,C 180,E1 15711.275,E2 15711.275} C_VEL
LIN {X 0,Y 295.893,Z 1131.616,A -85,B 0,C 180,E1 15718.518,E2 15718.518} C_VEL
LIN {X 0,Y 288.95,Z 1148.98,A -85,B 0,C 180,E1 15726.224,E2 15726.224} C_VEL
LIN {X 0,Y 285.17,Z 1161.721,A -85,B 0,C 180,E1 15734.658,E2 15734.658} C_VEL
LIN {X 0,Y 284.102,Z 1167.462,A -85,B 0,C 180,E1 15740.831,E2 15740.831} C_VEL
LIN {X 0,Y 283.935,Z 1170.312,A -85,B 0,C 180,E1 15746.954,E2 15746.954} C_VEL
LIN {X 0,Y 284.063,Z 1170.318,A -85,B 0,C 180,E1 15753.045,E2 15753.045} C_VEL
LIN {X 0,Y 284.339,Z 1165.856,A -85,B 0,C 180,E1 15761.166,E2 15761.166} C_VEL
LIN {X 0,Y 286.464,Z 1156.551,A -85,B 0,C 180,E1 15769.223,E2 15769.223} C_VEL
LIN {X 0,Y 291.288,Z 1142.635,A -85,B 0,C 180,E1 15776.955,E2 15776.955} C_VEL
LIN {X 0,Y 300.828,Z 1120.79,A -85,B 0,C 180,E1 15785.231,E2 15785.231} C_VEL
LIN {X 0,Y 313.764,Z 1093.708,A -85,B 0,C 180,E1 15792.324,E2 15792.324} C_VEL
LIN {X 0,Y 328.762,Z 1061.667,A -85,B 0,C 180,E1 15798.187,E2 15798.187} C_VEL
LIN {X 0,Y 343.464,Z 1026.704,A -85,B 0,C 180,E1 15802.7,E2 15802.7} C_VEL
LIN {X 0,Y 357.39,Z 987.583,A -85,B 0,C 180,E1 15806.191,E2 15806.191} C_VEL
LIN {X 0,Y 358.372,Z 984.389,A -85,B 0,C 180,E1 15806.411,E2 15806.411} C_VEL
LIN {X 0,Y 358.429,Z 977.969,A -85,B 0,C 180,E1 15807.309,E2 15807.309} C_VEL
LIN {X 0,Y 354.577,Z 970.018,A -85,B 0,C 180,E1 15809.378,E2 15809.378} C_VEL
LIN {X 0,Y 346.894,Z 947.416,A -85,B 0,C 180,E1 15814.836,E2 15814.836} C_VEL
LIN {X 0,Y 338.521,Z 928.431,A -85,B 0,C 180,E1 15820.969,E2 15820.969} C_VEL
LIN {X 0,Y 332.173,Z 916.536,A -85,B 0,C 180,E1 15826.577,E2 15826.577} C_VEL
LIN {X 0,Y 329.289,Z 911.054,A -85,B 0,C 180,E1 15830.105,E2 15830.105} C_VEL
LIN {X 0,Y 326.617,Z 905.142,A -85,B 0,C 180,E1 15835.362,E2 15835.362} C_VEL
LIN {X 0,Y 326.204,Z 904.978,A -85,B 0,C 180,E1 15844.643,E2 15844.643} C_VEL
LIN {X 0,Y 327,Z 907.212,A -85,B 0,C 180,E1 15847.124,E2 15847.124} C_VEL
LIN {X 0,Y 330.007,Z 913.495,A -85,B 0,C 180,E1 15852.293,E2 15852.293} C_VEL
LIN {X 0,Y 334.763,Z 923.097,A -85,B 0,C 180,E1 15857.502,E2 15857.502} C_VEL
LIN {X 0,Y 342.253,Z 940.721,A -85,B 0,C 180,E1 15864.068,E2 15864.068} C_VEL
LIN {X 0,Y 348.789,Z 960.506,A -85,B 0,C 180,E1 15869.48,E2 15869.48} C_VEL
LIN {X 0,Y 352.38,Z 978.652,A -85,B 0,C 180,E1 15873.475,E2 15873.475} C_VEL
LIN {X 0,Y 338.444,Z 1015.693,A -85,B 0,C 180,E1 15877.053,E2 15877.053} C_VEL
LIN {X 0,Y 323.928,Z 1048.094,A -85,B 0,C 180,E1 15881.485,E2 15881.485} C_VEL
LIN {X 0,Y 308.684,Z 1078.224,A -85,B 0,C 180,E1 15887.313,E2 15887.313} C_VEL
LIN {X 0,Y 295.196,Z 1103.758,A -85,B 0,C 180,E1 15894.435,E2 15894.435} C_VEL
LIN {X 0,Y 285.175,Z 1123.499,A -85,B 0,C 180,E1 15902.418,E2 15902.418} C_VEL
LIN {X 0,Y 279.249,Z 1137.706,A -85,B 0,C 180,E1 15911.081,E2 15911.081} C_VEL
LIN {X 0,Y 276.729,Z 1145.577,A -85,B 0,C 180,E1 15918.963,E2 15918.963} C_VEL
LIN {X 0,Y 276.059,Z 1149.353,A -85,B 0,C 180,E1 15926.866,E2 15926.866} C_VEL
LIN {X 0,Y 276.166,Z 1149.329,A -85,B 0,C 180,E1 15933.132,E2 15933.132} C_VEL
LIN {X 0,Y 276.762,Z 1145.475,A -85,B 0,C 180,E1 15941.072,E2 15941.072} C_VEL
LIN {X 0,Y 279.554,Z 1136.754,A -85,B 0,C 180,E1 15949.499,E2 15949.499} C_VEL
LIN {X 0,Y 286.044,Z 1121.656,A -85,B 0,C 180,E1 15958.345,E2 15958.345} C_VEL
LIN {X 0,Y 296.615,Z 1101.066,A -85,B 0,C 180,E1 15966.334,E2 15966.334} C_VEL
LIN {X 0,Y 309.674,Z 1076.244,A -85,B 0,C 180,E1 15973.038,E2 15973.038} C_VEL
LIN {X 0,Y 324.734,Z 1046.262,A -85,B 0,C 180,E1 15978.717,E2 15978.717} C_VEL
LIN {X 0,Y 340.041,Z 1011.728,A -85,B 0,C 180,E1 15983.306,E2 15983.306} C_VEL
LIN {X 0,Y 352.56,Z 977.246,A -85,B 0,C 180,E1 15986.595,E2 15986.595} C_VEL
LIN {X 0,Y 347.009,Z 954.917,A -85,B 0,C 180,E1 15991.812,E2 15991.812} C_VEL
LIN {X 0,Y 339.777,Z 934.601,A -85,B 0,C 180,E1 15997.844,E2 15997.844} C_VEL
LIN {X 0,Y 332.281,Z 917.64,A -85,B 0,C 180,E1 16004.87,E2 16004.87} C_VEL
LIN {X 0,Y 328.615,Z 910.815,A -85,B 0,C 180,E1 16009.416,E2 16009.416} C_VEL
LIN {X 0,Y 326.218,Z 905.037,A -85,B 0,C 180,E1 16014.692,E2 16014.692} C_VEL
LIN {X 0,Y 325.905,Z 904.702,A -85,B 0,C 180,E1 16023.318,E2 16023.318} C_VEL
LIN {X 0,Y 327.069,Z 906.449,A -85,B 0,C 180,E1 16026.291,E2 16026.291} C_VEL
LIN {X 0,Y 330.769,Z 913.733,A -85,B 0,C 180,E1 16031.93,E2 16031.93} C_VEL
LIN {X 0,Y 336.285,Z 924.002,A -85,B 0,C 180,E1 16037.329,E2 16037.329} C_VEL
LIN {X 0,Y 344.034,Z 940.666,A -85,B 0,C 180,E1 16043.25,E2 16043.25} C_VEL
LIN {X 0,Y 351.823,Z 961.169,A -85,B 0,C 180,E1 16048.654,E2 16048.654} C_VEL
LIN {X 0,Y 356.079,Z 977.279,A -85,B 0,C 180,E1 16052.052,E2 16052.052} C_VEL
LIN {X 0,Y 342.821,Z 1015.579,A -85,B 0,C 180,E1 16055.119,E2 16055.119} C_VEL
LIN {X 0,Y 327.41,Z 1052.222,A -85,B 0,C 180,E1 16059.38,E2 16059.38} C_VEL
LIN {X 0,Y 312.074,Z 1084.558,A -85,B 0,C 180,E1 16064.789,E2 16064.789} C_VEL
LIN {X 0,Y 298.152,Z 1112.522,A -85,B 0,C 180,E1 16071.463,E2 16071.463} C_VEL
LIN {X 0,Y 286.926,Z 1135.608,A -85,B 0,C 180,E1 16079.335,E2 16079.335} C_VEL
LIN {X 0,Y 279.975,Z 1152.623,A -85,B 0,C 180,E1 16087.835,E2 16087.835} C_VEL
LIN {X 0,Y 277.014,Z 1163.053,A -85,B 0,C 180,E1 16095.811,E2 16095.811} C_VEL
LIN {X 0,Y 275.979,Z 1168.943,A -85,B 0,C 180,E1 16103.722,E2 16103.722} C_VEL
LIN {X 0,Y 276.185,Z 1170.378,A -85,B 0,C 180,E1 16110,E2 16110} C_VEL
LIN {X 0,Y 276.003,Z 1168.947,A -85,B 0,C 180,E1 16116.278,E2 16116.278} C_VEL
LIN {X 0,Y 276.926,Z 1163.058,A -85,B 0,C 180,E1 16124.195,E2 16124.195} C_VEL
LIN {X 0,Y 279.964,Z 1152.64,A -85,B 0,C 180,E1 16132.167,E2 16132.167} C_VEL
LIN {X 0,Y 286.921,Z 1135.635,A -85,B 0,C 180,E1 16140.663,E2 16140.663} C_VEL
LIN {X 0,Y 298.007,Z 1112.689,A -85,B 0,C 180,E1 16148.512,E2 16148.512} C_VEL
LIN {X 0,Y 312.844,Z 1083.038,A -85,B 0,C 180,E1 16155.52,E2 16155.52} C_VEL
LIN {X 0,Y 328.434,Z 1050.265,A -85,B 0,C 180,E1 16160.885,E2 16160.885} C_VEL
LIN {X 0,Y 343.575,Z 1013.94,A -85,B 0,C 180,E1 16165.041,E2 16165.041} C_VEL
LIN {X 0,Y 356.154,Z 976.093,A -85,B 0,C 180,E1 16168.133,E2 16168.133} C_VEL
LIN {X 0,Y 354.577,Z 970.018,A -85,B 0,C 180,E1 16169.378,E2 16169.378} C_VEL
LIN {X 0,Y 350.912,Z 964.299,A -85,B 0,C 180,E1 16171.202,E2 16171.202} C_VEL
LIN {X 0,Y 344.02,Z 956.717,A -85,B 0,C 180,E1 16174.444,E2 16174.444} C_VEL
LIN {X 0,Y 337.182,Z 939.689,A -85,B 0,C 180,E1 16179.745,E2 16179.745} C_VEL
LIN {X 0,Y 330.596,Z 925.102,A -85,B 0,C 180,E1 16185.921,E2 16185.921} C_VEL
LIN {X 0,Y 326.913,Z 918.485,A -85,B 0,C 180,E1 16190.368,E2 16190.368} C_VEL
LIN {X 0,Y 324.72,Z 912.808,A -85,B 0,C 180,E1 16195.335,E2 16195.335} C_VEL
LIN {X 0,Y 323.998,Z 912.557,A -85,B 0,C 180,E1 16204.006,E2 16204.006} C_VEL
LIN {X 0,Y 324.683,Z 914.127,A -85,B 0,C 180,E1 16206.481,E2 16206.481} C_VEL
LIN {X 0,Y 327.584,Z 921.029,A -85,B 0,C 180,E1 16212.117,E2 16212.117} C_VEL
LIN {X 0,Y 332.314,Z 931.798,A -85,B 0,C 180,E1 16217.853,E2 16217.853} C_VEL
LIN {X 0,Y 338.85,Z 948.189,A -85,B 0,C 180,E1 16223.976,E2 16223.976} C_VEL
LIN {X 0,Y 344.539,Z 968.086,A -85,B 0,C 180,E1 16229.482,E2 16229.482} C_VEL
LIN {X 0,Y 346.84,Z 982.402,A -85,B 0,C 180,E1 16232.662,E2 16232.662} C_VEL
LIN {X 0,Y 332.703,Z 1018.155,A -85,B 0,C 180,E1 16236.203,E2 16236.203} C_VEL
LIN {X 0,Y 317.991,Z 1049.615,A -85,B 0,C 180,E1 16240.599,E2 16240.599} C_VEL
LIN {X 0,Y 302.733,Z 1078.528,A -85,B 0,C 180,E1 16246.266,E2 16246.266} C_VEL
LIN {X 0,Y 288.596,Z 1104.085,A -85,B 0,C 180,E1 16253.503,E2 16253.503} C_VEL
LIN {X 0,Y 277.964,Z 1123.804,A -85,B 0,C 180,E1 16261.639,E2 16261.639} C_VEL
LIN {X 0,Y 271.448,Z 1138.463,A -85,B 0,C 180,E1 16270.911,E2 16270.911} C_VEL
LIN {X 0,Y 268.885,Z 1145.876,A -85,B 0,C 180,E1 16278.636,E2 16278.636} C_VEL
LIN {X 0,Y 268.156,Z 1149.649,A -85,B 0,C 180,E1 16286.774,E2 16286.774} C_VEL
LIN {X 0,Y 268.26,Z 1149.626,A -85,B 0,C 180,E1 16293.224,E2 16293.224} C_VEL
LIN {X 0,Y 268.919,Z 1145.776,A -85,B 0,C 180,E1 16301.399,E2 16301.399} C_VEL
LIN {X 0,Y 271.648,Z 1137.873,A -85,B 0,C 180,E1 16309.469,E2 16309.469} C_VEL
LIN {X 0,Y 278.08,Z 1123.625,A -85,B 0,C 180,E1 16318.347,E2 16318.347} C_VEL
LIN {X 0,Y 289.366,Z 1102.746,A -85,B 0,C 180,E1 16326.849,E2 16326.849} C_VEL
LIN {X 0,Y 303.751,Z 1076.623,A -85,B 0,C 180,E1 16334.068,E2 16334.068} C_VEL
LIN {X 0,Y 319.793,Z 1045.849,A -85,B 0,C 180,E1 16339.919,E2 16339.919} C_VEL
LIN {X 0,Y 335.807,Z 1010.802,A -85,B 0,C 180,E1 16344.536,E2 16344.536} C_VEL
LIN {X 0,Y 347.072,Z 980.731,A -85,B 0,C 180,E1 16347.445,E2 16347.445} C_VEL
LIN {X 0,Y 342.065,Z 959.09,A -85,B 0,C 180,E1 16352.762,E2 16352.762} C_VEL
LIN {X 0,Y 336.109,Z 941.143,A -85,B 0,C 180,E1 16358.261,E2 16358.261} C_VEL
LIN {X 0,Y 329.68,Z 925.422,A -85,B 0,C 180,E1 16364.937,E2 16364.937} C_VEL
LIN {X 0,Y 326.179,Z 918.203,A -85,B 0,C 180,E1 16369.696,E2 16369.696} C_VEL
LIN {X 0,Y 324.234,Z 912.675,A -85,B 0,C 180,E1 16374.66,E2 16374.66} C_VEL
LIN {X 0,Y 324.009,Z 912.384,A -85,B 0,C 180,E1 16383.338,E2 16383.338} C_VEL
LIN {X 0,Y 325.023,Z 914.148,A -85,B 0,C 180,E1 16386.184,E2 16386.184} C_VEL
LIN {X 0,Y 328.326,Z 921.312,A -85,B 0,C 180,E1 16391.768,E2 16391.768} C_VEL
LIN {X 0,Y 333.414,Z 931.306,A -85,B 0,C 180,E1 16397.05,E2 16397.05} C_VEL
